{attribute 'Tc2GvlVarNames'}
VAR_GLOBAL

(*HORZ*)

	dwArm2HorzHomeStart 		: DWORD; (* %MD21900 *)
	dwArm2HorzHomeReset 		: DWORD; (* %MD21940 *)


(* xxx Horz SlantedLeft DWORD LINK with %MX21000-MX21099  xxx*)
(*======================================================*)

	dwArm2HorzStn1SlantedLeft 	: DWORD; (* %MD21004 *)
	dwArm2HorzStn2SlantedLeft 	: DWORD; (* %MD21008 *)
	dwArm2HorzStn3SlantedLeft 	: DWORD; (* %MD21012 *)
	dwArm2HorzStn4SlantedLeft 	: DWORD; (* %MD21016 *)
	dwArm2HorzStn5SlantedLeft 	: DWORD; (* %MD21020 *)
	dwArm2HorzStn6SlantedLeft 	: DWORD; (* %MD21024 *)
	dwArm2HorzStn7SlantedLeft 	: DWORD; (* %MD21028 *)
	dwArm2HorzStn8SlantedLeft 	: DWORD; (* %MD21032 *)
	dwArm2HorzStn9SlantedLeft 	: DWORD; (* %MD21036 *)
	dwArm2HorzStn10SlantedLeft 	: DWORD; (* %MD21040 *)
	dwArm2HorzStn11SlantedLeft 	: DWORD; (* %MD21044 *)
	dwArm2HorzStn12SlantedLeft 	: DWORD; (* %MD21048 *)

(* xxx Horz SlantedRight DWORD LINK with %MX21100-MX21199  xxx*)
(*======================================================*)

	dwArm2HorzStn1SlantedRight 	: DWORD; (* %MD21104 *)
	dwArm2HorzStn2SlantedRight 	: DWORD; (* %MD21108 *)
	dwArm2HorzStn3SlantedRight 	: DWORD; (* %MD21112 *)
	dwArm2HorzStn4SlantedRight 	: DWORD; (* %MD21116 *)
	dwArm2HorzStn5SlantedRight 	: DWORD; (* %MD21120 *)
	dwArm2HorzStn6SlantedRight 	: DWORD; (* %MD21124 *)
	dwArm2HorzStn7SlantedRight 	: DWORD; (* %MD21128 *)
	dwArm2HorzStn8SlantedRight 	: DWORD; (* %MD21132 *)
	dwArm2HorzStn9SlantedRight 	: DWORD; (* %MD21136 *)
	dwArm2HorzStn10SlantedRight 	: DWORD; (* %MD21140 *)
	dwArm2HorzStn11SlantedRight 	: DWORD; (* %MD21144 *)
	dwArm2HorzStn12SlantedRight 	: DWORD; (* %MD21148 *)

(* xxx Hook DWORD LINK with %MX21200-MX21299  xxx*)
(*======================================================*)

	dwArm2Ld1Hook 				: DWORD; (* %MD21252 *)
	dwArm2Uld1Hook 			: DWORD; (* %MD21256 *)
	dwArm2HorzStn1Hook 			: DWORD; (* %MD21204 *)
	dwArm2HorzStn2Hook 			: DWORD; (* %MD21208 *)
	dwArm2HorzStn3Hook 			: DWORD; (* %MD21212 *)
	dwArm2HorzStn4Hook 			: DWORD; (* %MD21216 *)
	dwArm2HorzStn5Hook 			: DWORD; (* %MD21220 *)
	dwArm2HorzStn6Hook 			: DWORD; (* %MD21224 *)
	dwArm2HorzStn7Hook 			: DWORD; (* %MD21228 *)
	dwArm2HorzStn8Hook 			: DWORD; (* %MD21232 *)
	dwArm2HorzStn9Hook 			: DWORD; (* %MD21236 *)
	dwArm2HorzStn10Hook 		: DWORD; (* %MD21240 *)
	dwArm2HorzStn11Hook 		: DWORD; (* %MD21244 *)
	dwArm2HorzStn12Hook 		: DWORD; (* %MD21248 *)

(* xxx Unhook DWORD LINK with %MX21300-MX21399  xxx*)
(*======================================================*)

	dwArm2Ld1Unhook 			: DWORD; (* %MD21352 *)
	dwArm2Uld1Unhook 			: DWORD; (* %MD21356 *)
	dwArm2HorzStn1Unhook 		: DWORD; (* %MD21304 *)
	dwArm2HorzStn2Unhook 		: DWORD; (* %MD21308 *)
	dwArm2HorzStn3Unhook 		: DWORD; (* %MD21312 *)
	dwArm2HorzStn4Unhook 		: DWORD; (* %MD21316 *)
	dwArm2HorzStn5Unhook 		: DWORD; (* %MD21320 *)
	dwArm2HorzStn6Unhook 		: DWORD; (* %MD21324 *)
	dwArm2HorzStn7Unhook 		: DWORD; (* %MD21328 *)
	dwArm2HorzStn8Unhook 		: DWORD; (* %MD21332 *)
	dwArm2HorzStn9Unhook 		: DWORD; (* %MD21336 *)
	dwArm2HorzStn10Unhook 		: DWORD; (* %MD21340 *)
	dwArm2HorzStn11Unhook 		: DWORD; (* %MD21344 *)
	dwArm2HorzStn12Unhook 		: DWORD; (* %MD21348 *)

(*VERT*)

	dwArm2VertHomeStart 			: DWORD; (* %MD26900 *)
	dwArm2VertHomeReset 		: DWORD; (* %MD26940 *)

(* xxx Up DWORD LINK with %MX26000-MX26099  xxx*)
(*======================================================*)

	dwArm2Ld1Up 				: DWORD; (* %MD26052 *)
	dwArm2Uld1Up 				: DWORD; (* %MD26056 *)
	dwArm2VertStn1Up 			: DWORD; (* %MD26004 *)
	dwArm2VertStn2Up 			: DWORD; (* %MD26008 *)
	dwArm2VertStn3Up 			: DWORD; (* %MD26012 *)
	dwArm2VertStn4Up 			: DWORD; (* %MD26016 *)
	dwArm2VertStn5Up 			: DWORD; (* %MD26020 *)
	dwArm2VertStn6Up 			: DWORD; (* %MD26024 *)
	dwArm2VertStn7Up 			: DWORD; (* %MD26028 *)
	dwArm2VertStn8Up 			: DWORD; (* %MD26032 *)
	dwArm2VertStn9Up 			: DWORD; (* %MD26036 *)
	dwArm2VertStn10Up 			: DWORD; (* %MD26040 *)
	dwArm2VertStn11Up 			: DWORD; (* %MD26044 *)
	dwArm2VertStn12Up 			: DWORD; (* %MD26048 *)

(* xxx Down SpSlanted DWORD LINK with %MX26100-MX26199  xxx*)
(*======================================================*)
(*Arm Mid Pos*)
	dwArm2VertStn1SpSlanted 		: DWORD; (* %MD26104 *)
	dwArm2VertStn2SpSlanted 		: DWORD; (* %MD26108 *)
	dwArm2VertStn3SpSlanted 		: DWORD; (* %MD26112 *)
	dwArm2VertStn4SpSlanted 		: DWORD; (* %MD26116 *)
	dwArm2VertStn5SpSlanted 		: DWORD; (* %MD26120 *)
	dwArm2VertStn6SpSlanted 		: DWORD; (* %MD26124 *)
	dwArm2VertStn7SpSlanted 		: DWORD; (* %MD26128 *)
	dwArm2VertStn8SpSlanted 		: DWORD; (* %MD26132 *)
	dwArm2VertStn9SpSlanted 		: DWORD; (* %MD26136 *)
	dwArm2VertStn10SpSlanted 	: DWORD; (* %MD26140 *)
	dwArm2VertStn11SpSlanted 	: DWORD; (* %MD26144 *)
	dwArm2VertStn12SpSlanted 	: DWORD; (* %MD26148 *)

(* xxx Down Regular DWORD LINK with %MX26200-MX26299  xxx*)
(*======================================================*)

	dwArm2VertStn1Regular 		: DWORD; (* %MD26204 *)
	dwArm2VertStn2Regular 		: DWORD; (* %MD26208 *)
	dwArm2VertStn3Regular 		: DWORD; (* %MD26212 *)
	dwArm2VertStn4Regular 		: DWORD; (* %MD26216 *)
	dwArm2VertStn5Regular 		: DWORD; (* %MD26220 *)
	dwArm2VertStn6Regular 		: DWORD; (* %MD26224 *)
	dwArm2VertStn7Regular 		: DWORD; (* %MD26228 *)
	dwArm2VertStn8Regular 		: DWORD; (* %MD26232 *)
	dwArm2VertStn9Regular 		: DWORD; (* %MD26236 *)
	dwArm2VertStn10Regular 		: DWORD; (* %MD26240 *)
	dwArm2VertStn11Regular 		: DWORD; (* %MD26244 *)
	dwArm2VertStn12Regular 		: DWORD; (* %MD26248 *)

(* xxx Up AgiUp DWORD LINK with %MX26300-MX26399  xxx*)
(*======================================================*)

	dwArm2VertStn1AglUp 			: DWORD; (* %MD26304 *)
	dwArm2VertStn2AglUp 			: DWORD; (* %MD26308 *)
	dwArm2VertStn3AglUp 			: DWORD; (* %MD26312 *)
	dwArm2VertStn4AglUp 			: DWORD; (* %MD26316 *)
	dwArm2VertStn5AglUp 			: DWORD; (* %MD26320 *)
	dwArm2VertStn6AglUp 			: DWORD; (* %MD26324 *)
	dwArm2VertStn7AglUp 			: DWORD; (* %MD26328 *)
	dwArm2VertStn8AglUp 			: DWORD; (* %MD26332 *)
	dwArm2VertStn9AglUp 			: DWORD; (* %MD26336 *)
	dwArm2VertStn10AglUp 		: DWORD; (* %MD26340 *)
	dwArm2VertStn11AglUp 		: DWORD; (* %MD26344 *)
	dwArm2VertStn12AglUp 		: DWORD; (* %MD26348 *)

(* xxx Down AgiDown DWORD LINK with %MX26400-MX26499  xxx*)
(*======================================================*)

	dwArm2VertStn1AglDown 		: DWORD; (* %MD26404 *)
	dwArm2VertStn2AglDown 		: DWORD; (* %MD26408 *)
	dwArm2VertStn3AglDown 		: DWORD; (* %MD26412 *)
	dwArm2VertStn4AglDown 		: DWORD; (* %MD26416 *)
	dwArm2VertStn5AglDown 		: DWORD; (* %MD26420 *)
	dwArm2VertStn6AglDown 		: DWORD; (* %MD26424 *)
	dwArm2VertStn7AglDown 		: DWORD; (* %MD26428 *)
	dwArm2VertStn8AglDown 		: DWORD; (* %MD26432 *)
	dwArm2VertStn9AglDown 		: DWORD; (* %MD26436 *)
	dwArm2VertStn10AglDown 		: DWORD; (* %MD26440 *)
	dwArm2VertStn11AglDown 		: DWORD; (* %MD26444 *)
	dwArm2VertStn12AglDown 		: DWORD; (* %MD26448 *)

(* xxx Down DWORD LINK with %MX26500-MX26599  xxx*)
(*======================================================*)

	dwArm2Ld1Down 				: DWORD; (* %MD26552 *)
	dwArm2Uld1Down 			: DWORD; (* %MD26556 *)
	dwArm2VertStn1Down 			: DWORD; (* %MD26504 *)
	dwArm2VertStn2Down 			: DWORD; (* %MD26508 *)
	dwArm2VertStn3Down 			: DWORD; (* %MD26512 *)
	dwArm2VertStn4Down 			: DWORD; (* %MD26516 *)
	dwArm2VertStn5Down 			: DWORD; (* %MD26520 *)
	dwArm2VertStn6Down 			: DWORD; (* %MD26524 *)
	dwArm2VertStn7Down 			: DWORD; (* %MD26528 *)
	dwArm2VertStn8Down 			: DWORD; (* %MD26532 *)
	dwArm2VertStn9Down 			: DWORD; (* %MD26536 *)
	dwArm2VertStn10Down 		: DWORD; (* %MD26540 *)
	dwArm2VertStn11Down 		: DWORD; (* %MD26544 *)
	dwArm2VertStn12Down 		: DWORD; (* %MD26548 *)

(*LIFTER*)

	dwSlowPull2LifterHomeStart 	: DWORD; (* %MD31900 *)
	dwSlowPull2LifterHomeReset 	: DWORD; (* %MD31940 *)

(* xxx Up/Down LifterUp DWORD LINK with %MX31000-   xxx*)
(*======================================================*)

	dwSlowPull2LifterStn1Up 		: DWORD; (* %MD31004 *)
	dwSlowPull2LifterStn2Up 		: DWORD; (* %MD31008 *)
	dwSlowPull2LifterStn3Up 		: DWORD; (* %MD31012 *)
	dwSlowPull2LifterStn4Up 		: DWORD; (* %MD31016 *)
	dwSlowPull2LifterStn5Up 		: DWORD; (* %MD31020 *)
	dwSlowPull2LifterStn6Up 		: DWORD; (* %MD31024 *)
	dwSlowPull2LifterStn7Up 		: DWORD; (* %MD31028 *)
	dwSlowPull2LifterStn8Up 		: DWORD; (* %MD31032 *)
	dwSlowPull2LifterStn9Up 		: DWORD; (* %MD31036 *)
	dwSlowPull2LifterStn10Up 		: DWORD; (* %MD31040 *)
	dwSlowPull2LifterStn11Up 		: DWORD; (* %MD31044 *)
	dwSlowPull2LifterStn12Up 		: DWORD; (* %MD31048 *)

(* xxx Up/Down LifterDown DWORD LINK with %MX31000-   xxx*)
(*======================================================*)

	dwSlowPull2LifterStn1Down 		: DWORD; (* %MD31304 *)
	dwSlowPull2LifterStn2Down 		: DWORD; (* %MD31308 *)
	dwSlowPull2LifterStn3Down 		: DWORD; (* %MD31312 *)
	dwSlowPull2LifterStn4Down 		: DWORD; (* %MD31316 *)
	dwSlowPull2LifterStn5Down 		: DWORD; (* %MD31320 *)
	dwSlowPull2LifterStn6Down 		: DWORD; (* %MD31324 *)
	dwSlowPull2LifterStn7Down 		: DWORD; (* %MD31328 *)
	dwSlowPull2LifterStn8Down 		: DWORD; (* %MD31332 *)
	dwSlowPull2LifterStn9Down 		: DWORD; (* %MD31336 *)
	dwSlowPull2LifterStn10Down 	: DWORD; (* %MD31340 *)
	dwSlowPull2LifterStn11Down 	: DWORD; (* %MD31344 *)
	dwSlowPull2LifterStn12Down 	: DWORD; (* %MD31348 *)

(* xxx Up/Down LifterAgiUp DWORD LINK with %MX31000-   xxx*)
(*======================================================*)

	dwSlowPull2LifterStn1AgiUp 	: DWORD; (* %MD31104 *)
	dwSlowPull2LifterStn2AgiUp 	: DWORD; (* %MD31108 *)
	dwSlowPull2LifterStn3AgiUp 	: DWORD; (* %MD31112 *)
	dwSlowPull2LifterStn4AgiUp 	: DWORD; (* %MD31116 *)
	dwSlowPull2LifterStn5AgiUp 	: DWORD; (* %MD31120 *)
	dwSlowPull2LifterStn6AgiUp 	: DWORD; (* %MD31124 *)
	dwSlowPull2LifterStn7AgiUp 	: DWORD; (* %MD31128 *)
	dwSlowPull2LifterStn8AgiUp 	: DWORD; (* %MD31132 *)
	dwSlowPull2LifterStn9AgiUp 	: DWORD; (* %MD31136 *)
	dwSlowPull2LifterStn10AgiUp 	: DWORD; (* %MD31140 *)
	dwSlowPull2LifterStn11AgiUp 	: DWORD; (* %MD31144 *)
	dwSlowPull2LifterStn12AgiUp 	: DWORD; (* %MD31148 *)

(* xxx Up/Down LifterAgiDown DWORD LINK with %MX31000-   xxx*)
(*======================================================*)

	dwSlowPull2LifterStn1AgiDown 	: DWORD; (* %MD31204 *)
	dwSlowPull2LifterStn2AgiDown 	: DWORD; (* %MD31208 *)
	dwSlowPull2LifterStn3AgiDown 	: DWORD; (* %MD31212 *)
	dwSlowPull2LifterStn4AgiDown 	: DWORD; (* %MD31216 *)
	dwSlowPull2LifterStn5AgiDown 	: DWORD; (* %MD31220 *)
	dwSlowPull2LifterStn6AgiDown 	: DWORD; (* %MD31224 *)
	dwSlowPull2LifterStn7AgiDown 	: DWORD; (* %MD31228 *)
	dwSlowPull2LifterStn8AgiDown 	: DWORD; (* %MD31232 *)
	dwSlowPull2LifterStn9AgiDown 	: DWORD; (* %MD31236 *)
	dwSlowPull2LifterStn10AgiDown 	: DWORD; (* %MD31240 *)
	dwSlowPull2LifterStn11AgiDown 	: DWORD; (* %MD31244 *)
	dwSlowPull2LifterStn12AgiDown 	: DWORD; (* %MD31248 *)

(* xxxxxxxxxxxxxxxxxxxxxxxxxxxxxxxxxxxxxxx Home xxxxxxxxxxxxxxxxxxxxxxxxxxxxxxxxxxxxxxx*)
(*====================== Vert Home BOOL LINK with %MX26900 ======================*)

	bArm2VertHomeStart_00 AT %MX26900.0 : BOOL;
	bArm2VertHomeStart_01 AT %MX26900.1 : BOOL;
	bArm2VertHomeStart_02 AT %MX26900.2 : BOOL;
	bArm2VertHomeStart_03 AT %MX26900.3 : BOOL;
	bArm2VertHomeStart_04 AT %MX26900.4 : BOOL;
	bArm2VertHomeStart_05 AT %MX26900.5 : BOOL;
	bArm2VertHomeStart_06 AT %MX26900.6 : BOOL;
	bArm2VertHomeStart_07 AT %MX26900.7 : BOOL;
	bArm2VertHomeStart_08 AT %MX26900.8 : BOOL;
	bArm2VertHomeStart_09 AT %MX26900.9 : BOOL;
	bArm2VertHomeStart_10 AT %MX26900.10 : BOOL;
	bArm2VertHomeStart_11 AT %MX26900.11 : BOOL;
	bArm2VertHomeStart_12 AT %MX26900.12 : BOOL;
	bArm2VertHomeStart_13 AT %MX26900.13 : BOOL;
	bArm2VertHomeStart_14 AT %MX26900.14 : BOOL;
	bArm2VertHomeStart_15 AT %MX26900.15 : BOOL;
	bArm2VertHomeStart_16 AT %MX26900.16 : BOOL;
	bArm2VertHomeStart_17 AT %MX26900.17 : BOOL;
	bArm2VertHomeStart_18 AT %MX26900.18 : BOOL;
	bArm2VertHomeStart_19 AT %MX26900.19 : BOOL;
	bArm2VertHomeStart_20 AT %MX26900.20 : BOOL;
	bArm2VertHomeStart_21 AT %MX26900.21 : BOOL;
	bArm2VertHomeStart_22 AT %MX26900.22 : BOOL;
	bArm2VertHomeStart_23 AT %MX26900.23 : BOOL;
	bArm2VertHomeStart_24 AT %MX26900.24 : BOOL;
	bArm2VertHomeStart_25 AT %MX26900.25 : BOOL;
	bArm2VertHomeStart_26 AT %MX26900.26 : BOOL;
	bArm2VertHomeStart_27 AT %MX26900.27 : BOOL;
	bArm2VertHomeStart_28 AT %MX26900.28 : BOOL;
	bArm2VertHomeStart_29 AT %MX26900.29 : BOOL;
	bArm2VertHomeStart_30 AT %MX26900.30 : BOOL;
	bArm2VertHomeStart_31 AT %MX26900.31 : BOOL;

	bArm2HorzHomeStart_00 AT %MX21900.0 : BOOL;
	bArm2HorzHomeStart_01 AT %MX21900.1 : BOOL;
	bArm2HorzHomeStart_02 AT %MX21900.2 : BOOL;
	bArm2HorzHomeStart_03 AT %MX21900.3 : BOOL;
	bArm2HorzHomeStart_04 AT %MX21900.4 : BOOL;
	bArm2HorzHomeStart_05 AT %MX21900.5 : BOOL;
	bArm2HorzHomeStart_06 AT %MX21900.6 : BOOL;
	bArm2HorzHomeStart_07 AT %MX21900.7 : BOOL;
	bArm2HorzHomeStart_08 AT %MX21900.8 : BOOL;
	bArm2HorzHomeStart_09 AT %MX21900.9 : BOOL;
	bArm2HorzHomeStart_10 AT %MX21900.10 : BOOL;
	bArm2HorzHomeStart_11 AT %MX21900.11 : BOOL;
	bArm2HorzHomeStart_12 AT %MX21900.12 : BOOL;
	bArm2HorzHomeStart_13 AT %MX21900.13 : BOOL;
	bArm2HorzHomeStart_14 AT %MX21900.14 : BOOL;
	bArm2HorzHomeStart_15 AT %MX21900.15 : BOOL;
	bArm2HorzHomeStart_16 AT %MX21900.16 : BOOL;
	bArm2HorzHomeStart_17 AT %MX21900.17 : BOOL;
	bArm2HorzHomeStart_18 AT %MX21900.18 : BOOL;
	bArm2HorzHomeStart_19 AT %MX21900.19 : BOOL;
	bArm2HorzHomeStart_20 AT %MX21900.20 : BOOL;
	bArm2HorzHomeStart_21 AT %MX21900.21 : BOOL;
	bArm2HorzHomeStart_22 AT %MX21900.22 : BOOL;
	bArm2HorzHomeStart_23 AT %MX21900.23 : BOOL;
	bArm2HorzHomeStart_24 AT %MX21900.24 : BOOL;
	bArm2HorzHomeStart_25 AT %MX21900.25 : BOOL;
	bArm2HorzHomeStart_26 AT %MX21900.26 : BOOL;
	bArm2HorzHomeStart_27 AT %MX21900.27 : BOOL;
	bArm2HorzHomeStart_28 AT %MX21900.28 : BOOL;
	bArm2HorzHomeStart_29 AT %MX21900.29 : BOOL;
	bArm2HorzHomeStart_30 AT %MX21900.30 : BOOL;
	bArm2HorzHomeStart_31 AT %MX21900.31 : BOOL;

	bSlowPull2LifterHomeStart_00 AT %MX31900.0 : BOOL;
	bSlowPull2LifterHomeStart_01 AT %MX31900.1 : BOOL;
	bSlowPull2LifterHomeStart_02 AT %MX31900.2 : BOOL;
	bSlowPull2LifterHomeStart_03 AT %MX31900.3 : BOOL;
	bSlowPull2LifterHomeStart_04 AT %MX31900.4 : BOOL;
	bSlowPull2LifterHomeStart_05 AT %MX31900.5 : BOOL;
	bSlowPull2LifterHomeStart_06 AT %MX31900.6 : BOOL;
	bSlowPull2LifterHomeStart_07 AT %MX31900.7 : BOOL;
	bSlowPull2LifterHomeStart_08 AT %MX31900.8 : BOOL;
	bSlowPull2LifterHomeStart_09 AT %MX31900.9 : BOOL;
	bSlowPull2LifterHomeStart_10 AT %MX31900.10 : BOOL;
	bSlowPull2LifterHomeStart_11 AT %MX31900.11 : BOOL;
	bSlowPull2LifterHomeStart_12 AT %MX31900.12 : BOOL;
	bSlowPull2LifterHomeStart_13 AT %MX31900.13 : BOOL;
	bSlowPull2LifterHomeStart_14 AT %MX31900.14 : BOOL;
	bSlowPull2LifterHomeStart_15 AT %MX31900.15 : BOOL;
	bSlowPull2LifterHomeStart_16 AT %MX31900.16 : BOOL;
	bSlowPull2LifterHomeStart_17 AT %MX31900.17 : BOOL;
	bSlowPull2LifterHomeStart_18 AT %MX31900.18 : BOOL;
	bSlowPull2LifterHomeStart_19 AT %MX31900.19 : BOOL;
	bSlowPull2LifterHomeStart_20 AT %MX31900.20 : BOOL;
	bSlowPull2LifterHomeStart_21 AT %MX31900.21 : BOOL;
	bSlowPull2LifterHomeStart_22 AT %MX31900.22 : BOOL;
	bSlowPull2LifterHomeStart_23 AT %MX31900.23 : BOOL;
	bSlowPull2LifterHomeStart_24 AT %MX31900.24 : BOOL;
	bSlowPull2LifterHomeStart_25 AT %MX31900.25 : BOOL;
	bSlowPull2LifterHomeStart_26 AT %MX31900.26 : BOOL;
	bSlowPull2LifterHomeStart_27 AT %MX31900.27 : BOOL;
	bSlowPull2LifterHomeStart_28 AT %MX31900.28 : BOOL;
	bSlowPull2LifterHomeStart_29 AT %MX31900.29 : BOOL;
	bSlowPull2LifterHomeStart_30 AT %MX31900.30 : BOOL;
	bSlowPull2LifterHomeStart_31 AT %MX31900.31 : BOOL;

(*=============================== SlantedLeft word ===============================*)
(*====================== SlantedLeft BOOL LINK with %MX21000-MX21099 ======================*)

	bArm2HorzStn1SlantedLeft_00 AT %MX21004.0 : BOOL;
	bArm2HorzStn1SlantedLeft_01 AT %MX21004.1 : BOOL;
	bArm2HorzStn1SlantedLeft_02 AT %MX21004.2 : BOOL;
	bArm2HorzStn1SlantedLeft_03 AT %MX21004.3 : BOOL;
	bArm2HorzStn1SlantedLeft_04 AT %MX21004.4 : BOOL;
	bArm2HorzStn1SlantedLeft_05 AT %MX21004.5 : BOOL;
	bArm2HorzStn1SlantedLeft_06 AT %MX21004.6 : BOOL;
	bArm2HorzStn1SlantedLeft_07 AT %MX21004.7 : BOOL;
	bArm2HorzStn1SlantedLeft_08 AT %MX21004.8 : BOOL;
	bArm2HorzStn1SlantedLeft_09 AT %MX21004.9 : BOOL;
	bArm2HorzStn1SlantedLeft_10 AT %MX21004.10 : BOOL;
	bArm2HorzStn1SlantedLeft_11 AT %MX21004.11 : BOOL;
	bArm2HorzStn1SlantedLeft_12 AT %MX21004.12 : BOOL;
	bArm2HorzStn1SlantedLeft_13 AT %MX21004.13 : BOOL;
	bArm2HorzStn1SlantedLeft_14 AT %MX21004.14 : BOOL;
	bArm2HorzStn1SlantedLeft_15 AT %MX21004.15 : BOOL;
	bArm2HorzStn1SlantedLeft_16 AT %MX21004.16 : BOOL;
	bArm2HorzStn1SlantedLeft_17 AT %MX21004.17 : BOOL;
	bArm2HorzStn1SlantedLeft_18 AT %MX21004.18 : BOOL;
	bArm2HorzStn1SlantedLeft_19 AT %MX21004.19 : BOOL;
	bArm2HorzStn1SlantedLeft_20 AT %MX21004.20 : BOOL;
	bArm2HorzStn1SlantedLeft_21 AT %MX21004.21 : BOOL;
	bArm2HorzStn1SlantedLeft_22 AT %MX21004.22 : BOOL;
	bArm2HorzStn1SlantedLeft_23 AT %MX21004.23 : BOOL;
	bArm2HorzStn1SlantedLeft_24 AT %MX21004.24 : BOOL;
	bArm2HorzStn1SlantedLeft_25 AT %MX21004.25 : BOOL;
	bArm2HorzStn1SlantedLeft_26 AT %MX21004.26 : BOOL;
	bArm2HorzStn1SlantedLeft_27 AT %MX21004.27 : BOOL;
	bArm2HorzStn1SlantedLeft_28 AT %MX21004.28 : BOOL;
	bArm2HorzStn1SlantedLeft_29 AT %MX21004.29 : BOOL;
	bArm2HorzStn1SlantedLeft_30 AT %MX21004.30 : BOOL;
	bArm2HorzStn1SlantedLeft_31 AT %MX21004.31 : BOOL;

	bArm2HorzStn2SlantedLeft_00 AT %MX21008.0 : BOOL;
	bArm2HorzStn2SlantedLeft_01 AT %MX21008.1 : BOOL;
	bArm2HorzStn2SlantedLeft_02 AT %MX21008.2 : BOOL;
	bArm2HorzStn2SlantedLeft_03 AT %MX21008.3 : BOOL;
	bArm2HorzStn2SlantedLeft_04 AT %MX21008.4 : BOOL;
	bArm2HorzStn2SlantedLeft_05 AT %MX21008.5 : BOOL;
	bArm2HorzStn2SlantedLeft_06 AT %MX21008.6 : BOOL;
	bArm2HorzStn2SlantedLeft_07 AT %MX21008.7 : BOOL;
	bArm2HorzStn2SlantedLeft_08 AT %MX21008.8 : BOOL;
	bArm2HorzStn2SlantedLeft_09 AT %MX21008.9 : BOOL;
	bArm2HorzStn2SlantedLeft_10 AT %MX21008.10 : BOOL;
	bArm2HorzStn2SlantedLeft_11 AT %MX21008.11 : BOOL;
	bArm2HorzStn2SlantedLeft_12 AT %MX21008.12 : BOOL;
	bArm2HorzStn2SlantedLeft_13 AT %MX21008.13 : BOOL;
	bArm2HorzStn2SlantedLeft_14 AT %MX21008.14 : BOOL;
	bArm2HorzStn2SlantedLeft_15 AT %MX21008.15 : BOOL;
	bArm2HorzStn2SlantedLeft_16 AT %MX21008.16 : BOOL;
	bArm2HorzStn2SlantedLeft_17 AT %MX21008.17 : BOOL;
	bArm2HorzStn2SlantedLeft_18 AT %MX21008.18 : BOOL;
	bArm2HorzStn2SlantedLeft_19 AT %MX21008.19 : BOOL;
	bArm2HorzStn2SlantedLeft_20 AT %MX21008.20 : BOOL;
	bArm2HorzStn2SlantedLeft_21 AT %MX21008.21 : BOOL;
	bArm2HorzStn2SlantedLeft_22 AT %MX21008.22 : BOOL;
	bArm2HorzStn2SlantedLeft_23 AT %MX21008.23 : BOOL;
	bArm2HorzStn2SlantedLeft_24 AT %MX21008.24 : BOOL;
	bArm2HorzStn2SlantedLeft_25 AT %MX21008.25 : BOOL;
	bArm2HorzStn2SlantedLeft_26 AT %MX21008.26 : BOOL;
	bArm2HorzStn2SlantedLeft_27 AT %MX21008.27 : BOOL;
	bArm2HorzStn2SlantedLeft_28 AT %MX21008.28 : BOOL;
	bArm2HorzStn2SlantedLeft_29 AT %MX21008.29 : BOOL;
	bArm2HorzStn2SlantedLeft_30 AT %MX21008.30 : BOOL;
	bArm2HorzStn2SlantedLeft_31 AT %MX21008.31 : BOOL;

	bArm2HorzStn3SlantedLeft_00 AT %MX21012.0 : BOOL;
	bArm2HorzStn3SlantedLeft_01 AT %MX21012.1 : BOOL;
	bArm2HorzStn3SlantedLeft_02 AT %MX21012.2 : BOOL;
	bArm2HorzStn3SlantedLeft_03 AT %MX21012.3 : BOOL;
	bArm2HorzStn3SlantedLeft_04 AT %MX21012.4 : BOOL;
	bArm2HorzStn3SlantedLeft_05 AT %MX21012.5 : BOOL;
	bArm2HorzStn3SlantedLeft_06 AT %MX21012.6 : BOOL;
	bArm2HorzStn3SlantedLeft_07 AT %MX21012.7 : BOOL;
	bArm2HorzStn3SlantedLeft_08 AT %MX21012.8 : BOOL;
	bArm2HorzStn3SlantedLeft_09 AT %MX21012.9 : BOOL;
	bArm2HorzStn3SlantedLeft_10 AT %MX21012.10 : BOOL;
	bArm2HorzStn3SlantedLeft_11 AT %MX21012.11 : BOOL;
	bArm2HorzStn3SlantedLeft_12 AT %MX21012.12 : BOOL;
	bArm2HorzStn3SlantedLeft_13 AT %MX21012.13 : BOOL;
	bArm2HorzStn3SlantedLeft_14 AT %MX21012.14 : BOOL;
	bArm2HorzStn3SlantedLeft_15 AT %MX21012.15 : BOOL;
	bArm2HorzStn3SlantedLeft_16 AT %MX21012.16 : BOOL;
	bArm2HorzStn3SlantedLeft_17 AT %MX21012.17 : BOOL;
	bArm2HorzStn3SlantedLeft_18 AT %MX21012.18 : BOOL;
	bArm2HorzStn3SlantedLeft_19 AT %MX21012.19 : BOOL;
	bArm2HorzStn3SlantedLeft_20 AT %MX21012.20 : BOOL;
	bArm2HorzStn3SlantedLeft_21 AT %MX21012.21 : BOOL;
	bArm2HorzStn3SlantedLeft_22 AT %MX21012.22 : BOOL;
	bArm2HorzStn3SlantedLeft_23 AT %MX21012.23 : BOOL;
	bArm2HorzStn3SlantedLeft_24 AT %MX21012.24 : BOOL;
	bArm2HorzStn3SlantedLeft_25 AT %MX21012.25 : BOOL;
	bArm2HorzStn3SlantedLeft_26 AT %MX21012.26 : BOOL;
	bArm2HorzStn3SlantedLeft_27 AT %MX21012.27 : BOOL;
	bArm2HorzStn3SlantedLeft_28 AT %MX21012.28 : BOOL;
	bArm2HorzStn3SlantedLeft_29 AT %MX21012.29 : BOOL;
	bArm2HorzStn3SlantedLeft_30 AT %MX21012.30 : BOOL;
	bArm2HorzStn3SlantedLeft_31 AT %MX21012.31 : BOOL;

	bArm2HorzStn4SlantedLeft_00 AT %MX21016.0 : BOOL;
	bArm2HorzStn4SlantedLeft_01 AT %MX21016.1 : BOOL;
	bArm2HorzStn4SlantedLeft_02 AT %MX21016.2 : BOOL;
	bArm2HorzStn4SlantedLeft_03 AT %MX21016.3 : BOOL;
	bArm2HorzStn4SlantedLeft_04 AT %MX21016.4 : BOOL;
	bArm2HorzStn4SlantedLeft_05 AT %MX21016.5 : BOOL;
	bArm2HorzStn4SlantedLeft_06 AT %MX21016.6 : BOOL;
	bArm2HorzStn4SlantedLeft_07 AT %MX21016.7 : BOOL;
	bArm2HorzStn4SlantedLeft_08 AT %MX21016.8 : BOOL;
	bArm2HorzStn4SlantedLeft_09 AT %MX21016.9 : BOOL;
	bArm2HorzStn4SlantedLeft_10 AT %MX21016.10 : BOOL;
	bArm2HorzStn4SlantedLeft_11 AT %MX21016.11 : BOOL;
	bArm2HorzStn4SlantedLeft_12 AT %MX21016.12 : BOOL;
	bArm2HorzStn4SlantedLeft_13 AT %MX21016.13 : BOOL;
	bArm2HorzStn4SlantedLeft_14 AT %MX21016.14 : BOOL;
	bArm2HorzStn4SlantedLeft_15 AT %MX21016.15 : BOOL;
	bArm2HorzStn4SlantedLeft_16 AT %MX21016.16 : BOOL;
	bArm2HorzStn4SlantedLeft_17 AT %MX21016.17 : BOOL;
	bArm2HorzStn4SlantedLeft_18 AT %MX21016.18 : BOOL;
	bArm2HorzStn4SlantedLeft_19 AT %MX21016.19 : BOOL;
	bArm2HorzStn4SlantedLeft_20 AT %MX21016.20 : BOOL;
	bArm2HorzStn4SlantedLeft_21 AT %MX21016.21 : BOOL;
	bArm2HorzStn4SlantedLeft_22 AT %MX21016.22 : BOOL;
	bArm2HorzStn4SlantedLeft_23 AT %MX21016.23 : BOOL;
	bArm2HorzStn4SlantedLeft_24 AT %MX21016.24 : BOOL;
	bArm2HorzStn4SlantedLeft_25 AT %MX21016.25 : BOOL;
	bArm2HorzStn4SlantedLeft_26 AT %MX21016.26 : BOOL;
	bArm2HorzStn4SlantedLeft_27 AT %MX21016.27 : BOOL;
	bArm2HorzStn4SlantedLeft_28 AT %MX21016.28 : BOOL;
	bArm2HorzStn4SlantedLeft_29 AT %MX21016.29 : BOOL;
	bArm2HorzStn4SlantedLeft_30 AT %MX21016.30 : BOOL;
	bArm2HorzStn4SlantedLeft_31 AT %MX21016.31 : BOOL;

	bArm2HorzStn5SlantedLeft_00 AT %MX21020.0 : BOOL;
	bArm2HorzStn5SlantedLeft_01 AT %MX21020.1 : BOOL;
	bArm2HorzStn5SlantedLeft_02 AT %MX21020.2 : BOOL;
	bArm2HorzStn5SlantedLeft_03 AT %MX21020.3 : BOOL;
	bArm2HorzStn5SlantedLeft_04 AT %MX21020.4 : BOOL;
	bArm2HorzStn5SlantedLeft_05 AT %MX21020.5 : BOOL;
	bArm2HorzStn5SlantedLeft_06 AT %MX21020.6 : BOOL;
	bArm2HorzStn5SlantedLeft_07 AT %MX21020.7 : BOOL;
	bArm2HorzStn5SlantedLeft_08 AT %MX21020.8 : BOOL;
	bArm2HorzStn5SlantedLeft_09 AT %MX21020.9 : BOOL;
	bArm2HorzStn5SlantedLeft_10 AT %MX21020.10 : BOOL;
	bArm2HorzStn5SlantedLeft_11 AT %MX21020.11 : BOOL;
	bArm2HorzStn5SlantedLeft_12 AT %MX21020.12 : BOOL;
	bArm2HorzStn5SlantedLeft_13 AT %MX21020.13 : BOOL;
	bArm2HorzStn5SlantedLeft_14 AT %MX21020.14 : BOOL;
	bArm2HorzStn5SlantedLeft_15 AT %MX21020.15 : BOOL;
	bArm2HorzStn5SlantedLeft_16 AT %MX21020.16 : BOOL;
	bArm2HorzStn5SlantedLeft_17 AT %MX21020.17 : BOOL;
	bArm2HorzStn5SlantedLeft_18 AT %MX21020.18 : BOOL;
	bArm2HorzStn5SlantedLeft_19 AT %MX21020.19 : BOOL;
	bArm2HorzStn5SlantedLeft_20 AT %MX21020.20 : BOOL;
	bArm2HorzStn5SlantedLeft_21 AT %MX21020.21 : BOOL;
	bArm2HorzStn5SlantedLeft_22 AT %MX21020.22 : BOOL;
	bArm2HorzStn5SlantedLeft_23 AT %MX21020.23 : BOOL;
	bArm2HorzStn5SlantedLeft_24 AT %MX21020.24 : BOOL;
	bArm2HorzStn5SlantedLeft_25 AT %MX21020.25 : BOOL;
	bArm2HorzStn5SlantedLeft_26 AT %MX21020.26 : BOOL;
	bArm2HorzStn5SlantedLeft_27 AT %MX21020.27 : BOOL;
	bArm2HorzStn5SlantedLeft_28 AT %MX21020.28 : BOOL;
	bArm2HorzStn5SlantedLeft_29 AT %MX21020.29 : BOOL;
	bArm2HorzStn5SlantedLeft_30 AT %MX21020.30 : BOOL;
	bArm2HorzStn5SlantedLeft_31 AT %MX21020.31 : BOOL;

	bArm2HorzStn6SlantedLeft_00 AT %MX21024.0 : BOOL;
	bArm2HorzStn6SlantedLeft_01 AT %MX21024.1 : BOOL;
	bArm2HorzStn6SlantedLeft_02 AT %MX21024.2 : BOOL;
	bArm2HorzStn6SlantedLeft_03 AT %MX21024.3 : BOOL;
	bArm2HorzStn6SlantedLeft_04 AT %MX21024.4 : BOOL;
	bArm2HorzStn6SlantedLeft_05 AT %MX21024.5 : BOOL;
	bArm2HorzStn6SlantedLeft_06 AT %MX21024.6 : BOOL;
	bArm2HorzStn6SlantedLeft_07 AT %MX21024.7 : BOOL;
	bArm2HorzStn6SlantedLeft_08 AT %MX21024.8 : BOOL;
	bArm2HorzStn6SlantedLeft_09 AT %MX21024.9 : BOOL;
	bArm2HorzStn6SlantedLeft_10 AT %MX21024.10 : BOOL;
	bArm2HorzStn6SlantedLeft_11 AT %MX21024.11 : BOOL;
	bArm2HorzStn6SlantedLeft_12 AT %MX21024.12 : BOOL;
	bArm2HorzStn6SlantedLeft_13 AT %MX21024.13 : BOOL;
	bArm2HorzStn6SlantedLeft_14 AT %MX21024.14 : BOOL;
	bArm2HorzStn6SlantedLeft_15 AT %MX21024.15 : BOOL;
	bArm2HorzStn6SlantedLeft_16 AT %MX21024.16 : BOOL;
	bArm2HorzStn6SlantedLeft_17 AT %MX21024.17 : BOOL;
	bArm2HorzStn6SlantedLeft_18 AT %MX21024.18 : BOOL;
	bArm2HorzStn6SlantedLeft_19 AT %MX21024.19 : BOOL;
	bArm2HorzStn6SlantedLeft_20 AT %MX21024.20 : BOOL;
	bArm2HorzStn6SlantedLeft_21 AT %MX21024.21 : BOOL;
	bArm2HorzStn6SlantedLeft_22 AT %MX21024.22 : BOOL;
	bArm2HorzStn6SlantedLeft_23 AT %MX21024.23 : BOOL;
	bArm2HorzStn6SlantedLeft_24 AT %MX21024.24 : BOOL;
	bArm2HorzStn6SlantedLeft_25 AT %MX21024.25 : BOOL;
	bArm2HorzStn6SlantedLeft_26 AT %MX21024.26 : BOOL;
	bArm2HorzStn6SlantedLeft_27 AT %MX21024.27 : BOOL;
	bArm2HorzStn6SlantedLeft_28 AT %MX21024.28 : BOOL;
	bArm2HorzStn6SlantedLeft_29 AT %MX21024.29 : BOOL;
	bArm2HorzStn6SlantedLeft_30 AT %MX21024.30 : BOOL;
	bArm2HorzStn6SlantedLeft_31 AT %MX21024.31 : BOOL;

	bArm2HorzStn7SlantedLeft_00 AT %MX21028.0 : BOOL;
	bArm2HorzStn7SlantedLeft_01 AT %MX21028.1 : BOOL;
	bArm2HorzStn7SlantedLeft_02 AT %MX21028.2 : BOOL;
	bArm2HorzStn7SlantedLeft_03 AT %MX21028.3 : BOOL;
	bArm2HorzStn7SlantedLeft_04 AT %MX21028.4 : BOOL;
	bArm2HorzStn7SlantedLeft_05 AT %MX21028.5 : BOOL;
	bArm2HorzStn7SlantedLeft_06 AT %MX21028.6 : BOOL;
	bArm2HorzStn7SlantedLeft_07 AT %MX21028.7 : BOOL;
	bArm2HorzStn7SlantedLeft_08 AT %MX21028.8 : BOOL;
	bArm2HorzStn7SlantedLeft_09 AT %MX21028.9 : BOOL;
	bArm2HorzStn7SlantedLeft_10 AT %MX21028.10 : BOOL;
	bArm2HorzStn7SlantedLeft_11 AT %MX21028.11 : BOOL;
	bArm2HorzStn7SlantedLeft_12 AT %MX21028.12 : BOOL;
	bArm2HorzStn7SlantedLeft_13 AT %MX21028.13 : BOOL;
	bArm2HorzStn7SlantedLeft_14 AT %MX21028.14 : BOOL;
	bArm2HorzStn7SlantedLeft_15 AT %MX21028.15 : BOOL;
	bArm2HorzStn7SlantedLeft_16 AT %MX21028.16 : BOOL;
	bArm2HorzStn7SlantedLeft_17 AT %MX21028.17 : BOOL;
	bArm2HorzStn7SlantedLeft_18 AT %MX21028.18 : BOOL;
	bArm2HorzStn7SlantedLeft_19 AT %MX21028.19 : BOOL;
	bArm2HorzStn7SlantedLeft_20 AT %MX21028.20 : BOOL;
	bArm2HorzStn7SlantedLeft_21 AT %MX21028.21 : BOOL;
	bArm2HorzStn7SlantedLeft_22 AT %MX21028.22 : BOOL;
	bArm2HorzStn7SlantedLeft_23 AT %MX21028.23 : BOOL;
	bArm2HorzStn7SlantedLeft_24 AT %MX21028.24 : BOOL;
	bArm2HorzStn7SlantedLeft_25 AT %MX21028.25 : BOOL;
	bArm2HorzStn7SlantedLeft_26 AT %MX21028.26 : BOOL;
	bArm2HorzStn7SlantedLeft_27 AT %MX21028.27 : BOOL;
	bArm2HorzStn7SlantedLeft_28 AT %MX21028.28 : BOOL;
	bArm2HorzStn7SlantedLeft_29 AT %MX21028.29 : BOOL;
	bArm2HorzStn7SlantedLeft_30 AT %MX21028.30 : BOOL;
	bArm2HorzStn7SlantedLeft_31 AT %MX21028.31 : BOOL;

	bArm2HorzStn8SlantedLeft_00 AT %MX21032.0 : BOOL;
	bArm2HorzStn8SlantedLeft_01 AT %MX21032.1 : BOOL;
	bArm2HorzStn8SlantedLeft_02 AT %MX21032.2 : BOOL;
	bArm2HorzStn8SlantedLeft_03 AT %MX21032.3 : BOOL;
	bArm2HorzStn8SlantedLeft_04 AT %MX21032.4 : BOOL;
	bArm2HorzStn8SlantedLeft_05 AT %MX21032.5 : BOOL;
	bArm2HorzStn8SlantedLeft_06 AT %MX21032.6 : BOOL;
	bArm2HorzStn8SlantedLeft_07 AT %MX21032.7 : BOOL;
	bArm2HorzStn8SlantedLeft_08 AT %MX21032.8 : BOOL;
	bArm2HorzStn8SlantedLeft_09 AT %MX21032.9 : BOOL;
	bArm2HorzStn8SlantedLeft_10 AT %MX21032.10 : BOOL;
	bArm2HorzStn8SlantedLeft_11 AT %MX21032.11 : BOOL;
	bArm2HorzStn8SlantedLeft_12 AT %MX21032.12 : BOOL;
	bArm2HorzStn8SlantedLeft_13 AT %MX21032.13 : BOOL;
	bArm2HorzStn8SlantedLeft_14 AT %MX21032.14 : BOOL;
	bArm2HorzStn8SlantedLeft_15 AT %MX21032.15 : BOOL;
	bArm2HorzStn8SlantedLeft_16 AT %MX21032.16 : BOOL;
	bArm2HorzStn8SlantedLeft_17 AT %MX21032.17 : BOOL;
	bArm2HorzStn8SlantedLeft_18 AT %MX21032.18 : BOOL;
	bArm2HorzStn8SlantedLeft_19 AT %MX21032.19 : BOOL;
	bArm2HorzStn8SlantedLeft_20 AT %MX21032.20 : BOOL;
	bArm2HorzStn8SlantedLeft_21 AT %MX21032.21 : BOOL;
	bArm2HorzStn8SlantedLeft_22 AT %MX21032.22 : BOOL;
	bArm2HorzStn8SlantedLeft_23 AT %MX21032.23 : BOOL;
	bArm2HorzStn8SlantedLeft_24 AT %MX21032.24 : BOOL;
	bArm2HorzStn8SlantedLeft_25 AT %MX21032.25 : BOOL;
	bArm2HorzStn8SlantedLeft_26 AT %MX21032.26 : BOOL;
	bArm2HorzStn8SlantedLeft_27 AT %MX21032.27 : BOOL;
	bArm2HorzStn8SlantedLeft_28 AT %MX21032.28 : BOOL;
	bArm2HorzStn8SlantedLeft_29 AT %MX21032.29 : BOOL;
	bArm2HorzStn8SlantedLeft_30 AT %MX21032.30 : BOOL;
	bArm2HorzStn8SlantedLeft_31 AT %MX21032.31 : BOOL;

	bArm2HorzStn9SlantedLeft_00 AT %MX21036.0 : BOOL;
	bArm2HorzStn9SlantedLeft_01 AT %MX21036.1 : BOOL;
	bArm2HorzStn9SlantedLeft_02 AT %MX21036.2 : BOOL;
	bArm2HorzStn9SlantedLeft_03 AT %MX21036.3 : BOOL;
	bArm2HorzStn9SlantedLeft_04 AT %MX21036.4 : BOOL;
	bArm2HorzStn9SlantedLeft_05 AT %MX21036.5 : BOOL;
	bArm2HorzStn9SlantedLeft_06 AT %MX21036.6 : BOOL;
	bArm2HorzStn9SlantedLeft_07 AT %MX21036.7 : BOOL;
	bArm2HorzStn9SlantedLeft_08 AT %MX21036.8 : BOOL;
	bArm2HorzStn9SlantedLeft_09 AT %MX21036.9 : BOOL;
	bArm2HorzStn9SlantedLeft_10 AT %MX21036.10 : BOOL;
	bArm2HorzStn9SlantedLeft_11 AT %MX21036.11 : BOOL;
	bArm2HorzStn9SlantedLeft_12 AT %MX21036.12 : BOOL;
	bArm2HorzStn9SlantedLeft_13 AT %MX21036.13 : BOOL;
	bArm2HorzStn9SlantedLeft_14 AT %MX21036.14 : BOOL;
	bArm2HorzStn9SlantedLeft_15 AT %MX21036.15 : BOOL;
	bArm2HorzStn9SlantedLeft_16 AT %MX21036.16 : BOOL;
	bArm2HorzStn9SlantedLeft_17 AT %MX21036.17 : BOOL;
	bArm2HorzStn9SlantedLeft_18 AT %MX21036.18 : BOOL;
	bArm2HorzStn9SlantedLeft_19 AT %MX21036.19 : BOOL;
	bArm2HorzStn9SlantedLeft_20 AT %MX21036.20 : BOOL;
	bArm2HorzStn9SlantedLeft_21 AT %MX21036.21 : BOOL;
	bArm2HorzStn9SlantedLeft_22 AT %MX21036.22 : BOOL;
	bArm2HorzStn9SlantedLeft_23 AT %MX21036.23 : BOOL;
	bArm2HorzStn9SlantedLeft_24 AT %MX21036.24 : BOOL;
	bArm2HorzStn9SlantedLeft_25 AT %MX21036.25 : BOOL;
	bArm2HorzStn9SlantedLeft_26 AT %MX21036.26 : BOOL;
	bArm2HorzStn9SlantedLeft_27 AT %MX21036.27 : BOOL;
	bArm2HorzStn9SlantedLeft_28 AT %MX21036.28 : BOOL;
	bArm2HorzStn9SlantedLeft_29 AT %MX21036.29 : BOOL;
	bArm2HorzStn9SlantedLeft_30 AT %MX21036.30 : BOOL;
	bArm2HorzStn9SlantedLeft_31 AT %MX21036.31 : BOOL;

	bArm2HorzStn10SlantedLeft_00 AT %MX21040.0 : BOOL;
	bArm2HorzStn10SlantedLeft_01 AT %MX21040.1 : BOOL;
	bArm2HorzStn10SlantedLeft_02 AT %MX21040.2 : BOOL;
	bArm2HorzStn10SlantedLeft_03 AT %MX21040.3 : BOOL;
	bArm2HorzStn10SlantedLeft_04 AT %MX21040.4 : BOOL;
	bArm2HorzStn10SlantedLeft_05 AT %MX21040.5 : BOOL;
	bArm2HorzStn10SlantedLeft_06 AT %MX21040.6 : BOOL;
	bArm2HorzStn10SlantedLeft_07 AT %MX21040.7 : BOOL;
	bArm2HorzStn10SlantedLeft_08 AT %MX21040.8 : BOOL;
	bArm2HorzStn10SlantedLeft_09 AT %MX21040.9 : BOOL;
	bArm2HorzStn10SlantedLeft_10 AT %MX21040.10 : BOOL;
	bArm2HorzStn10SlantedLeft_11 AT %MX21040.11 : BOOL;
	bArm2HorzStn10SlantedLeft_12 AT %MX21040.12 : BOOL;
	bArm2HorzStn10SlantedLeft_13 AT %MX21040.13 : BOOL;
	bArm2HorzStn10SlantedLeft_14 AT %MX21040.14 : BOOL;
	bArm2HorzStn10SlantedLeft_15 AT %MX21040.15 : BOOL;
	bArm2HorzStn10SlantedLeft_16 AT %MX21040.16 : BOOL;
	bArm2HorzStn10SlantedLeft_17 AT %MX21040.17 : BOOL;
	bArm2HorzStn10SlantedLeft_18 AT %MX21040.18 : BOOL;
	bArm2HorzStn10SlantedLeft_19 AT %MX21040.19 : BOOL;
	bArm2HorzStn10SlantedLeft_20 AT %MX21040.20 : BOOL;
	bArm2HorzStn10SlantedLeft_21 AT %MX21040.21 : BOOL;
	bArm2HorzStn10SlantedLeft_22 AT %MX21040.22 : BOOL;
	bArm2HorzStn10SlantedLeft_23 AT %MX21040.23 : BOOL;
	bArm2HorzStn10SlantedLeft_24 AT %MX21040.24 : BOOL;
	bArm2HorzStn10SlantedLeft_25 AT %MX21040.25 : BOOL;
	bArm2HorzStn10SlantedLeft_26 AT %MX21040.26 : BOOL;
	bArm2HorzStn10SlantedLeft_27 AT %MX21040.27 : BOOL;
	bArm2HorzStn10SlantedLeft_28 AT %MX21040.28 : BOOL;
	bArm2HorzStn10SlantedLeft_29 AT %MX21040.29 : BOOL;
	bArm2HorzStn10SlantedLeft_30 AT %MX21040.30 : BOOL;
	bArm2HorzStn10SlantedLeft_31 AT %MX21040.31 : BOOL;

	bArm2HorzStn11SlantedLeft_00 AT %MX21044.0 : BOOL;
	bArm2HorzStn11SlantedLeft_01 AT %MX21044.1 : BOOL;
	bArm2HorzStn11SlantedLeft_02 AT %MX21044.2 : BOOL;
	bArm2HorzStn11SlantedLeft_03 AT %MX21044.3 : BOOL;
	bArm2HorzStn11SlantedLeft_04 AT %MX21044.4 : BOOL;
	bArm2HorzStn11SlantedLeft_05 AT %MX21044.5 : BOOL;
	bArm2HorzStn11SlantedLeft_06 AT %MX21044.6 : BOOL;
	bArm2HorzStn11SlantedLeft_07 AT %MX21044.7 : BOOL;
	bArm2HorzStn11SlantedLeft_08 AT %MX21044.8 : BOOL;
	bArm2HorzStn11SlantedLeft_09 AT %MX21044.9 : BOOL;
	bArm2HorzStn11SlantedLeft_10 AT %MX21044.10 : BOOL;
	bArm2HorzStn11SlantedLeft_11 AT %MX21044.11 : BOOL;
	bArm2HorzStn11SlantedLeft_12 AT %MX21044.12 : BOOL;
	bArm2HorzStn11SlantedLeft_13 AT %MX21044.13 : BOOL;
	bArm2HorzStn11SlantedLeft_14 AT %MX21044.14 : BOOL;
	bArm2HorzStn11SlantedLeft_15 AT %MX21044.15 : BOOL;
	bArm2HorzStn11SlantedLeft_16 AT %MX21044.16 : BOOL;
	bArm2HorzStn11SlantedLeft_17 AT %MX21044.17 : BOOL;
	bArm2HorzStn11SlantedLeft_18 AT %MX21044.18 : BOOL;
	bArm2HorzStn11SlantedLeft_19 AT %MX21044.19 : BOOL;
	bArm2HorzStn11SlantedLeft_20 AT %MX21044.20 : BOOL;
	bArm2HorzStn11SlantedLeft_21 AT %MX21044.21 : BOOL;
	bArm2HorzStn11SlantedLeft_22 AT %MX21044.22 : BOOL;
	bArm2HorzStn11SlantedLeft_23 AT %MX21044.23 : BOOL;
	bArm2HorzStn11SlantedLeft_24 AT %MX21044.24 : BOOL;
	bArm2HorzStn11SlantedLeft_25 AT %MX21044.25 : BOOL;
	bArm2HorzStn11SlantedLeft_26 AT %MX21044.26 : BOOL;
	bArm2HorzStn11SlantedLeft_27 AT %MX21044.27 : BOOL;
	bArm2HorzStn11SlantedLeft_28 AT %MX21044.28 : BOOL;
	bArm2HorzStn11SlantedLeft_29 AT %MX21044.29 : BOOL;
	bArm2HorzStn11SlantedLeft_30 AT %MX21044.30 : BOOL;
	bArm2HorzStn11SlantedLeft_31 AT %MX21044.31 : BOOL;

	bArm2HorzStn12SlantedLeft_00 AT %MX21048.0 : BOOL;
	bArm2HorzStn12SlantedLeft_01 AT %MX21048.1 : BOOL;
	bArm2HorzStn12SlantedLeft_02 AT %MX21048.2 : BOOL;
	bArm2HorzStn12SlantedLeft_03 AT %MX21048.3 : BOOL;
	bArm2HorzStn12SlantedLeft_04 AT %MX21048.4 : BOOL;
	bArm2HorzStn12SlantedLeft_05 AT %MX21048.5 : BOOL;
	bArm2HorzStn12SlantedLeft_06 AT %MX21048.6 : BOOL;
	bArm2HorzStn12SlantedLeft_07 AT %MX21048.7 : BOOL;
	bArm2HorzStn12SlantedLeft_08 AT %MX21048.8 : BOOL;
	bArm2HorzStn12SlantedLeft_09 AT %MX21048.9 : BOOL;
	bArm2HorzStn12SlantedLeft_10 AT %MX21048.10 : BOOL;
	bArm2HorzStn12SlantedLeft_11 AT %MX21048.11 : BOOL;
	bArm2HorzStn12SlantedLeft_12 AT %MX21048.12 : BOOL;
	bArm2HorzStn12SlantedLeft_13 AT %MX21048.13 : BOOL;
	bArm2HorzStn12SlantedLeft_14 AT %MX21048.14 : BOOL;
	bArm2HorzStn12SlantedLeft_15 AT %MX21048.15 : BOOL;
	bArm2HorzStn12SlantedLeft_16 AT %MX21048.16 : BOOL;
	bArm2HorzStn12SlantedLeft_17 AT %MX21048.17 : BOOL;
	bArm2HorzStn12SlantedLeft_18 AT %MX21048.18 : BOOL;
	bArm2HorzStn12SlantedLeft_19 AT %MX21048.19 : BOOL;
	bArm2HorzStn12SlantedLeft_20 AT %MX21048.20 : BOOL;
	bArm2HorzStn12SlantedLeft_21 AT %MX21048.21 : BOOL;
	bArm2HorzStn12SlantedLeft_22 AT %MX21048.22 : BOOL;
	bArm2HorzStn12SlantedLeft_23 AT %MX21048.23 : BOOL;
	bArm2HorzStn12SlantedLeft_24 AT %MX21048.24 : BOOL;
	bArm2HorzStn12SlantedLeft_25 AT %MX21048.25 : BOOL;
	bArm2HorzStn12SlantedLeft_26 AT %MX21048.26 : BOOL;
	bArm2HorzStn12SlantedLeft_27 AT %MX21048.27 : BOOL;
	bArm2HorzStn12SlantedLeft_28 AT %MX21048.28 : BOOL;
	bArm2HorzStn12SlantedLeft_29 AT %MX21048.29 : BOOL;
	bArm2HorzStn12SlantedLeft_30 AT %MX21048.30 : BOOL;
	bArm2HorzStn12SlantedLeft_31 AT %MX21048.31 : BOOL;


(*=============================== SlantedRight word ===============================*)
(*====================== SlantedRight BOOL LINK with %MX21100-MX21199 ======================*)

	bArm2HorzStn1SlantedRight_00 AT %MX21104.0 : BOOL;
	bArm2HorzStn1SlantedRight_01 AT %MX21104.1 : BOOL;
	bArm2HorzStn1SlantedRight_02 AT %MX21104.2 : BOOL;
	bArm2HorzStn1SlantedRight_03 AT %MX21104.3 : BOOL;
	bArm2HorzStn1SlantedRight_04 AT %MX21104.4 : BOOL;
	bArm2HorzStn1SlantedRight_05 AT %MX21104.5 : BOOL;
	bArm2HorzStn1SlantedRight_06 AT %MX21104.6 : BOOL;
	bArm2HorzStn1SlantedRight_07 AT %MX21104.7 : BOOL;
	bArm2HorzStn1SlantedRight_08 AT %MX21104.8 : BOOL;
	bArm2HorzStn1SlantedRight_09 AT %MX21104.9 : BOOL;
	bArm2HorzStn1SlantedRight_10 AT %MX21104.10 : BOOL;
	bArm2HorzStn1SlantedRight_11 AT %MX21104.11 : BOOL;
	bArm2HorzStn1SlantedRight_12 AT %MX21104.12 : BOOL;
	bArm2HorzStn1SlantedRight_13 AT %MX21104.13 : BOOL;
	bArm2HorzStn1SlantedRight_14 AT %MX21104.14 : BOOL;
	bArm2HorzStn1SlantedRight_15 AT %MX21104.15 : BOOL;
	bArm2HorzStn1SlantedRight_16 AT %MX21104.16 : BOOL;
	bArm2HorzStn1SlantedRight_17 AT %MX21104.17 : BOOL;
	bArm2HorzStn1SlantedRight_18 AT %MX21104.18 : BOOL;
	bArm2HorzStn1SlantedRight_19 AT %MX21104.19 : BOOL;
	bArm2HorzStn1SlantedRight_20 AT %MX21104.20 : BOOL;
	bArm2HorzStn1SlantedRight_21 AT %MX21104.21 : BOOL;
	bArm2HorzStn1SlantedRight_22 AT %MX21104.22 : BOOL;
	bArm2HorzStn1SlantedRight_23 AT %MX21104.23 : BOOL;
	bArm2HorzStn1SlantedRight_24 AT %MX21104.24 : BOOL;
	bArm2HorzStn1SlantedRight_25 AT %MX21104.25 : BOOL;
	bArm2HorzStn1SlantedRight_26 AT %MX21104.26 : BOOL;
	bArm2HorzStn1SlantedRight_27 AT %MX21104.27 : BOOL;
	bArm2HorzStn1SlantedRight_28 AT %MX21104.28 : BOOL;
	bArm2HorzStn1SlantedRight_29 AT %MX21104.29 : BOOL;
	bArm2HorzStn1SlantedRight_30 AT %MX21104.30 : BOOL;
	bArm2HorzStn1SlantedRight_31 AT %MX21104.31 : BOOL;

	bArm2HorzStn2SlantedRight_00 AT %MX21108.0 : BOOL;
	bArm2HorzStn2SlantedRight_01 AT %MX21108.1 : BOOL;
	bArm2HorzStn2SlantedRight_02 AT %MX21108.2 : BOOL;
	bArm2HorzStn2SlantedRight_03 AT %MX21108.3 : BOOL;
	bArm2HorzStn2SlantedRight_04 AT %MX21108.4 : BOOL;
	bArm2HorzStn2SlantedRight_05 AT %MX21108.5 : BOOL;
	bArm2HorzStn2SlantedRight_06 AT %MX21108.6 : BOOL;
	bArm2HorzStn2SlantedRight_07 AT %MX21108.7 : BOOL;
	bArm2HorzStn2SlantedRight_08 AT %MX21108.8 : BOOL;
	bArm2HorzStn2SlantedRight_09 AT %MX21108.9 : BOOL;
	bArm2HorzStn2SlantedRight_10 AT %MX21108.10 : BOOL;
	bArm2HorzStn2SlantedRight_11 AT %MX21108.11 : BOOL;
	bArm2HorzStn2SlantedRight_12 AT %MX21108.12 : BOOL;
	bArm2HorzStn2SlantedRight_13 AT %MX21108.13 : BOOL;
	bArm2HorzStn2SlantedRight_14 AT %MX21108.14 : BOOL;
	bArm2HorzStn2SlantedRight_15 AT %MX21108.15 : BOOL;
	bArm2HorzStn2SlantedRight_16 AT %MX21108.16 : BOOL;
	bArm2HorzStn2SlantedRight_17 AT %MX21108.17 : BOOL;
	bArm2HorzStn2SlantedRight_18 AT %MX21108.18 : BOOL;
	bArm2HorzStn2SlantedRight_19 AT %MX21108.19 : BOOL;
	bArm2HorzStn2SlantedRight_20 AT %MX21108.20 : BOOL;
	bArm2HorzStn2SlantedRight_21 AT %MX21108.21 : BOOL;
	bArm2HorzStn2SlantedRight_22 AT %MX21108.22 : BOOL;
	bArm2HorzStn2SlantedRight_23 AT %MX21108.23 : BOOL;
	bArm2HorzStn2SlantedRight_24 AT %MX21108.24 : BOOL;
	bArm2HorzStn2SlantedRight_25 AT %MX21108.25 : BOOL;
	bArm2HorzStn2SlantedRight_26 AT %MX21108.26 : BOOL;
	bArm2HorzStn2SlantedRight_27 AT %MX21108.27 : BOOL;
	bArm2HorzStn2SlantedRight_28 AT %MX21108.28 : BOOL;
	bArm2HorzStn2SlantedRight_29 AT %MX21108.29 : BOOL;
	bArm2HorzStn2SlantedRight_30 AT %MX21108.30 : BOOL;
	bArm2HorzStn2SlantedRight_31 AT %MX21108.31 : BOOL;

	bArm2HorzStn3SlantedRight_00 AT %MX21112.0 : BOOL;
	bArm2HorzStn3SlantedRight_01 AT %MX21112.1 : BOOL;
	bArm2HorzStn3SlantedRight_02 AT %MX21112.2 : BOOL;
	bArm2HorzStn3SlantedRight_03 AT %MX21112.3 : BOOL;
	bArm2HorzStn3SlantedRight_04 AT %MX21112.4 : BOOL;
	bArm2HorzStn3SlantedRight_05 AT %MX21112.5 : BOOL;
	bArm2HorzStn3SlantedRight_06 AT %MX21112.6 : BOOL;
	bArm2HorzStn3SlantedRight_07 AT %MX21112.7 : BOOL;
	bArm2HorzStn3SlantedRight_08 AT %MX21112.8 : BOOL;
	bArm2HorzStn3SlantedRight_09 AT %MX21112.9 : BOOL;
	bArm2HorzStn3SlantedRight_10 AT %MX21112.10 : BOOL;
	bArm2HorzStn3SlantedRight_11 AT %MX21112.11 : BOOL;
	bArm2HorzStn3SlantedRight_12 AT %MX21112.12 : BOOL;
	bArm2HorzStn3SlantedRight_13 AT %MX21112.13 : BOOL;
	bArm2HorzStn3SlantedRight_14 AT %MX21112.14 : BOOL;
	bArm2HorzStn3SlantedRight_15 AT %MX21112.15 : BOOL;
	bArm2HorzStn3SlantedRight_16 AT %MX21112.16 : BOOL;
	bArm2HorzStn3SlantedRight_17 AT %MX21112.17 : BOOL;
	bArm2HorzStn3SlantedRight_18 AT %MX21112.18 : BOOL;
	bArm2HorzStn3SlantedRight_19 AT %MX21112.19 : BOOL;
	bArm2HorzStn3SlantedRight_20 AT %MX21112.20 : BOOL;
	bArm2HorzStn3SlantedRight_21 AT %MX21112.21 : BOOL;
	bArm2HorzStn3SlantedRight_22 AT %MX21112.22 : BOOL;
	bArm2HorzStn3SlantedRight_23 AT %MX21112.23 : BOOL;
	bArm2HorzStn3SlantedRight_24 AT %MX21112.24 : BOOL;
	bArm2HorzStn3SlantedRight_25 AT %MX21112.25 : BOOL;
	bArm2HorzStn3SlantedRight_26 AT %MX21112.26 : BOOL;
	bArm2HorzStn3SlantedRight_27 AT %MX21112.27 : BOOL;
	bArm2HorzStn3SlantedRight_28 AT %MX21112.28 : BOOL;
	bArm2HorzStn3SlantedRight_29 AT %MX21112.29 : BOOL;
	bArm2HorzStn3SlantedRight_30 AT %MX21112.30 : BOOL;
	bArm2HorzStn3SlantedRight_31 AT %MX21112.31 : BOOL;

	bArm2HorzStn4SlantedRight_00 AT %MX21116.0 : BOOL;
	bArm2HorzStn4SlantedRight_01 AT %MX21116.1 : BOOL;
	bArm2HorzStn4SlantedRight_02 AT %MX21116.2 : BOOL;
	bArm2HorzStn4SlantedRight_03 AT %MX21116.3 : BOOL;
	bArm2HorzStn4SlantedRight_04 AT %MX21116.4 : BOOL;
	bArm2HorzStn4SlantedRight_05 AT %MX21116.5 : BOOL;
	bArm2HorzStn4SlantedRight_06 AT %MX21116.6 : BOOL;
	bArm2HorzStn4SlantedRight_07 AT %MX21116.7 : BOOL;
	bArm2HorzStn4SlantedRight_08 AT %MX21116.8 : BOOL;
	bArm2HorzStn4SlantedRight_09 AT %MX21116.9 : BOOL;
	bArm2HorzStn4SlantedRight_10 AT %MX21116.10 : BOOL;
	bArm2HorzStn4SlantedRight_11 AT %MX21116.11 : BOOL;
	bArm2HorzStn4SlantedRight_12 AT %MX21116.12 : BOOL;
	bArm2HorzStn4SlantedRight_13 AT %MX21116.13 : BOOL;
	bArm2HorzStn4SlantedRight_14 AT %MX21116.14 : BOOL;
	bArm2HorzStn4SlantedRight_15 AT %MX21116.15 : BOOL;
	bArm2HorzStn4SlantedRight_16 AT %MX21116.16 : BOOL;
	bArm2HorzStn4SlantedRight_17 AT %MX21116.17 : BOOL;
	bArm2HorzStn4SlantedRight_18 AT %MX21116.18 : BOOL;
	bArm2HorzStn4SlantedRight_19 AT %MX21116.19 : BOOL;
	bArm2HorzStn4SlantedRight_20 AT %MX21116.20 : BOOL;
	bArm2HorzStn4SlantedRight_21 AT %MX21116.21 : BOOL;
	bArm2HorzStn4SlantedRight_22 AT %MX21116.22 : BOOL;
	bArm2HorzStn4SlantedRight_23 AT %MX21116.23 : BOOL;
	bArm2HorzStn4SlantedRight_24 AT %MX21116.24 : BOOL;
	bArm2HorzStn4SlantedRight_25 AT %MX21116.25 : BOOL;
	bArm2HorzStn4SlantedRight_26 AT %MX21116.26 : BOOL;
	bArm2HorzStn4SlantedRight_27 AT %MX21116.27 : BOOL;
	bArm2HorzStn4SlantedRight_28 AT %MX21116.28 : BOOL;
	bArm2HorzStn4SlantedRight_29 AT %MX21116.29 : BOOL;
	bArm2HorzStn4SlantedRight_30 AT %MX21116.30 : BOOL;
	bArm2HorzStn4SlantedRight_31 AT %MX21116.31 : BOOL;

	bArm2HorzStn5SlantedRight_00 AT %MX21120.0 : BOOL;
	bArm2HorzStn5SlantedRight_01 AT %MX21120.1 : BOOL;
	bArm2HorzStn5SlantedRight_02 AT %MX21120.2 : BOOL;
	bArm2HorzStn5SlantedRight_03 AT %MX21120.3 : BOOL;
	bArm2HorzStn5SlantedRight_04 AT %MX21120.4 : BOOL;
	bArm2HorzStn5SlantedRight_05 AT %MX21120.5 : BOOL;
	bArm2HorzStn5SlantedRight_06 AT %MX21120.6 : BOOL;
	bArm2HorzStn5SlantedRight_07 AT %MX21120.7 : BOOL;
	bArm2HorzStn5SlantedRight_08 AT %MX21120.8 : BOOL;
	bArm2HorzStn5SlantedRight_09 AT %MX21120.9 : BOOL;
	bArm2HorzStn5SlantedRight_10 AT %MX21120.10 : BOOL;
	bArm2HorzStn5SlantedRight_11 AT %MX21120.11 : BOOL;
	bArm2HorzStn5SlantedRight_12 AT %MX21120.12 : BOOL;
	bArm2HorzStn5SlantedRight_13 AT %MX21120.13 : BOOL;
	bArm2HorzStn5SlantedRight_14 AT %MX21120.14 : BOOL;
	bArm2HorzStn5SlantedRight_15 AT %MX21120.15 : BOOL;
	bArm2HorzStn5SlantedRight_16 AT %MX21120.16 : BOOL;
	bArm2HorzStn5SlantedRight_17 AT %MX21120.17 : BOOL;
	bArm2HorzStn5SlantedRight_18 AT %MX21120.18 : BOOL;
	bArm2HorzStn5SlantedRight_19 AT %MX21120.19 : BOOL;
	bArm2HorzStn5SlantedRight_20 AT %MX21120.20 : BOOL;
	bArm2HorzStn5SlantedRight_21 AT %MX21120.21 : BOOL;
	bArm2HorzStn5SlantedRight_22 AT %MX21120.22 : BOOL;
	bArm2HorzStn5SlantedRight_23 AT %MX21120.23 : BOOL;
	bArm2HorzStn5SlantedRight_24 AT %MX21120.24 : BOOL;
	bArm2HorzStn5SlantedRight_25 AT %MX21120.25 : BOOL;
	bArm2HorzStn5SlantedRight_26 AT %MX21120.26 : BOOL;
	bArm2HorzStn5SlantedRight_27 AT %MX21120.27 : BOOL;
	bArm2HorzStn5SlantedRight_28 AT %MX21120.28 : BOOL;
	bArm2HorzStn5SlantedRight_29 AT %MX21120.29 : BOOL;
	bArm2HorzStn5SlantedRight_30 AT %MX21120.30 : BOOL;
	bArm2HorzStn5SlantedRight_31 AT %MX21120.31 : BOOL;

	bArm2HorzStn6SlantedRight_00 AT %MX21124.0 : BOOL;
	bArm2HorzStn6SlantedRight_01 AT %MX21124.1 : BOOL;
	bArm2HorzStn6SlantedRight_02 AT %MX21124.2 : BOOL;
	bArm2HorzStn6SlantedRight_03 AT %MX21124.3 : BOOL;
	bArm2HorzStn6SlantedRight_04 AT %MX21124.4 : BOOL;
	bArm2HorzStn6SlantedRight_05 AT %MX21124.5 : BOOL;
	bArm2HorzStn6SlantedRight_06 AT %MX21124.6 : BOOL;
	bArm2HorzStn6SlantedRight_07 AT %MX21124.7 : BOOL;
	bArm2HorzStn6SlantedRight_08 AT %MX21124.8 : BOOL;
	bArm2HorzStn6SlantedRight_09 AT %MX21124.9 : BOOL;
	bArm2HorzStn6SlantedRight_10 AT %MX21124.10 : BOOL;
	bArm2HorzStn6SlantedRight_11 AT %MX21124.11 : BOOL;
	bArm2HorzStn6SlantedRight_12 AT %MX21124.12 : BOOL;
	bArm2HorzStn6SlantedRight_13 AT %MX21124.13 : BOOL;
	bArm2HorzStn6SlantedRight_14 AT %MX21124.14 : BOOL;
	bArm2HorzStn6SlantedRight_15 AT %MX21124.15 : BOOL;
	bArm2HorzStn6SlantedRight_16 AT %MX21124.16 : BOOL;
	bArm2HorzStn6SlantedRight_17 AT %MX21124.17 : BOOL;
	bArm2HorzStn6SlantedRight_18 AT %MX21124.18 : BOOL;
	bArm2HorzStn6SlantedRight_19 AT %MX21124.19 : BOOL;
	bArm2HorzStn6SlantedRight_20 AT %MX21124.20 : BOOL;
	bArm2HorzStn6SlantedRight_21 AT %MX21124.21 : BOOL;
	bArm2HorzStn6SlantedRight_22 AT %MX21124.22 : BOOL;
	bArm2HorzStn6SlantedRight_23 AT %MX21124.23 : BOOL;
	bArm2HorzStn6SlantedRight_24 AT %MX21124.24 : BOOL;
	bArm2HorzStn6SlantedRight_25 AT %MX21124.25 : BOOL;
	bArm2HorzStn6SlantedRight_26 AT %MX21124.26 : BOOL;
	bArm2HorzStn6SlantedRight_27 AT %MX21124.27 : BOOL;
	bArm2HorzStn6SlantedRight_28 AT %MX21124.28 : BOOL;
	bArm2HorzStn6SlantedRight_29 AT %MX21124.29 : BOOL;
	bArm2HorzStn6SlantedRight_30 AT %MX21124.30 : BOOL;
	bArm2HorzStn6SlantedRight_31 AT %MX21124.31 : BOOL;

	bArm2HorzStn7SlantedRight_00 AT %MX21128.0 : BOOL;
	bArm2HorzStn7SlantedRight_01 AT %MX21128.1 : BOOL;
	bArm2HorzStn7SlantedRight_02 AT %MX21128.2 : BOOL;
	bArm2HorzStn7SlantedRight_03 AT %MX21128.3 : BOOL;
	bArm2HorzStn7SlantedRight_04 AT %MX21128.4 : BOOL;
	bArm2HorzStn7SlantedRight_05 AT %MX21128.5 : BOOL;
	bArm2HorzStn7SlantedRight_06 AT %MX21128.6 : BOOL;
	bArm2HorzStn7SlantedRight_07 AT %MX21128.7 : BOOL;
	bArm2HorzStn7SlantedRight_08 AT %MX21128.8 : BOOL;
	bArm2HorzStn7SlantedRight_09 AT %MX21128.9 : BOOL;
	bArm2HorzStn7SlantedRight_10 AT %MX21128.10 : BOOL;
	bArm2HorzStn7SlantedRight_11 AT %MX21128.11 : BOOL;
	bArm2HorzStn7SlantedRight_12 AT %MX21128.12 : BOOL;
	bArm2HorzStn7SlantedRight_13 AT %MX21128.13 : BOOL;
	bArm2HorzStn7SlantedRight_14 AT %MX21128.14 : BOOL;
	bArm2HorzStn7SlantedRight_15 AT %MX21128.15 : BOOL;
	bArm2HorzStn7SlantedRight_16 AT %MX21128.16 : BOOL;
	bArm2HorzStn7SlantedRight_17 AT %MX21128.17 : BOOL;
	bArm2HorzStn7SlantedRight_18 AT %MX21128.18 : BOOL;
	bArm2HorzStn7SlantedRight_19 AT %MX21128.19 : BOOL;
	bArm2HorzStn7SlantedRight_20 AT %MX21128.20 : BOOL;
	bArm2HorzStn7SlantedRight_21 AT %MX21128.21 : BOOL;
	bArm2HorzStn7SlantedRight_22 AT %MX21128.22 : BOOL;
	bArm2HorzStn7SlantedRight_23 AT %MX21128.23 : BOOL;
	bArm2HorzStn7SlantedRight_24 AT %MX21128.24 : BOOL;
	bArm2HorzStn7SlantedRight_25 AT %MX21128.25 : BOOL;
	bArm2HorzStn7SlantedRight_26 AT %MX21128.26 : BOOL;
	bArm2HorzStn7SlantedRight_27 AT %MX21128.27 : BOOL;
	bArm2HorzStn7SlantedRight_28 AT %MX21128.28 : BOOL;
	bArm2HorzStn7SlantedRight_29 AT %MX21128.29 : BOOL;
	bArm2HorzStn7SlantedRight_30 AT %MX21128.30 : BOOL;
	bArm2HorzStn7SlantedRight_31 AT %MX21128.31 : BOOL;

	bArm2HorzStn8SlantedRight_00 AT %MX21132.0 : BOOL;
	bArm2HorzStn8SlantedRight_01 AT %MX21132.1 : BOOL;
	bArm2HorzStn8SlantedRight_02 AT %MX21132.2 : BOOL;
	bArm2HorzStn8SlantedRight_03 AT %MX21132.3 : BOOL;
	bArm2HorzStn8SlantedRight_04 AT %MX21132.4 : BOOL;
	bArm2HorzStn8SlantedRight_05 AT %MX21132.5 : BOOL;
	bArm2HorzStn8SlantedRight_06 AT %MX21132.6 : BOOL;
	bArm2HorzStn8SlantedRight_07 AT %MX21132.7 : BOOL;
	bArm2HorzStn8SlantedRight_08 AT %MX21132.8 : BOOL;
	bArm2HorzStn8SlantedRight_09 AT %MX21132.9 : BOOL;
	bArm2HorzStn8SlantedRight_10 AT %MX21132.10 : BOOL;
	bArm2HorzStn8SlantedRight_11 AT %MX21132.11 : BOOL;
	bArm2HorzStn8SlantedRight_12 AT %MX21132.12 : BOOL;
	bArm2HorzStn8SlantedRight_13 AT %MX21132.13 : BOOL;
	bArm2HorzStn8SlantedRight_14 AT %MX21132.14 : BOOL;
	bArm2HorzStn8SlantedRight_15 AT %MX21132.15 : BOOL;
	bArm2HorzStn8SlantedRight_16 AT %MX21132.16 : BOOL;
	bArm2HorzStn8SlantedRight_17 AT %MX21132.17 : BOOL;
	bArm2HorzStn8SlantedRight_18 AT %MX21132.18 : BOOL;
	bArm2HorzStn8SlantedRight_19 AT %MX21132.19 : BOOL;
	bArm2HorzStn8SlantedRight_20 AT %MX21132.20 : BOOL;
	bArm2HorzStn8SlantedRight_21 AT %MX21132.21 : BOOL;
	bArm2HorzStn8SlantedRight_22 AT %MX21132.22 : BOOL;
	bArm2HorzStn8SlantedRight_23 AT %MX21132.23 : BOOL;
	bArm2HorzStn8SlantedRight_24 AT %MX21132.24 : BOOL;
	bArm2HorzStn8SlantedRight_25 AT %MX21132.25 : BOOL;
	bArm2HorzStn8SlantedRight_26 AT %MX21132.26 : BOOL;
	bArm2HorzStn8SlantedRight_27 AT %MX21132.27 : BOOL;
	bArm2HorzStn8SlantedRight_28 AT %MX21132.28 : BOOL;
	bArm2HorzStn8SlantedRight_29 AT %MX21132.29 : BOOL;
	bArm2HorzStn8SlantedRight_30 AT %MX21132.30 : BOOL;
	bArm2HorzStn8SlantedRight_31 AT %MX21132.31 : BOOL;

	bArm2HorzStn9SlantedRight_00 AT %MX21136.0 : BOOL;
	bArm2HorzStn9SlantedRight_01 AT %MX21136.1 : BOOL;
	bArm2HorzStn9SlantedRight_02 AT %MX21136.2 : BOOL;
	bArm2HorzStn9SlantedRight_03 AT %MX21136.3 : BOOL;
	bArm2HorzStn9SlantedRight_04 AT %MX21136.4 : BOOL;
	bArm2HorzStn9SlantedRight_05 AT %MX21136.5 : BOOL;
	bArm2HorzStn9SlantedRight_06 AT %MX21136.6 : BOOL;
	bArm2HorzStn9SlantedRight_07 AT %MX21136.7 : BOOL;
	bArm2HorzStn9SlantedRight_08 AT %MX21136.8 : BOOL;
	bArm2HorzStn9SlantedRight_09 AT %MX21136.9 : BOOL;
	bArm2HorzStn9SlantedRight_10 AT %MX21136.10 : BOOL;
	bArm2HorzStn9SlantedRight_11 AT %MX21136.11 : BOOL;
	bArm2HorzStn9SlantedRight_12 AT %MX21136.12 : BOOL;
	bArm2HorzStn9SlantedRight_13 AT %MX21136.13 : BOOL;
	bArm2HorzStn9SlantedRight_14 AT %MX21136.14 : BOOL;
	bArm2HorzStn9SlantedRight_15 AT %MX21136.15 : BOOL;
	bArm2HorzStn9SlantedRight_16 AT %MX21136.16 : BOOL;
	bArm2HorzStn9SlantedRight_17 AT %MX21136.17 : BOOL;
	bArm2HorzStn9SlantedRight_18 AT %MX21136.18 : BOOL;
	bArm2HorzStn9SlantedRight_19 AT %MX21136.19 : BOOL;
	bArm2HorzStn9SlantedRight_20 AT %MX21136.20 : BOOL;
	bArm2HorzStn9SlantedRight_21 AT %MX21136.21 : BOOL;
	bArm2HorzStn9SlantedRight_22 AT %MX21136.22 : BOOL;
	bArm2HorzStn9SlantedRight_23 AT %MX21136.23 : BOOL;
	bArm2HorzStn9SlantedRight_24 AT %MX21136.24 : BOOL;
	bArm2HorzStn9SlantedRight_25 AT %MX21136.25 : BOOL;
	bArm2HorzStn9SlantedRight_26 AT %MX21136.26 : BOOL;
	bArm2HorzStn9SlantedRight_27 AT %MX21136.27 : BOOL;
	bArm2HorzStn9SlantedRight_28 AT %MX21136.28 : BOOL;
	bArm2HorzStn9SlantedRight_29 AT %MX21136.29 : BOOL;
	bArm2HorzStn9SlantedRight_30 AT %MX21136.30 : BOOL;
	bArm2HorzStn9SlantedRight_31 AT %MX21136.31 : BOOL;

	bArm2HorzStn10SlantedRight_00 AT %MX21140.0 : BOOL;
	bArm2HorzStn10SlantedRight_01 AT %MX21140.1 : BOOL;
	bArm2HorzStn10SlantedRight_02 AT %MX21140.2 : BOOL;
	bArm2HorzStn10SlantedRight_03 AT %MX21140.3 : BOOL;
	bArm2HorzStn10SlantedRight_04 AT %MX21140.4 : BOOL;
	bArm2HorzStn10SlantedRight_05 AT %MX21140.5 : BOOL;
	bArm2HorzStn10SlantedRight_06 AT %MX21140.6 : BOOL;
	bArm2HorzStn10SlantedRight_07 AT %MX21140.7 : BOOL;
	bArm2HorzStn10SlantedRight_08 AT %MX21140.8 : BOOL;
	bArm2HorzStn10SlantedRight_09 AT %MX21140.9 : BOOL;
	bArm2HorzStn10SlantedRight_10 AT %MX21140.10 : BOOL;
	bArm2HorzStn10SlantedRight_11 AT %MX21140.11 : BOOL;
	bArm2HorzStn10SlantedRight_12 AT %MX21140.12 : BOOL;
	bArm2HorzStn10SlantedRight_13 AT %MX21140.13 : BOOL;
	bArm2HorzStn10SlantedRight_14 AT %MX21140.14 : BOOL;
	bArm2HorzStn10SlantedRight_15 AT %MX21140.15 : BOOL;
	bArm2HorzStn10SlantedRight_16 AT %MX21140.16 : BOOL;
	bArm2HorzStn10SlantedRight_17 AT %MX21140.17 : BOOL;
	bArm2HorzStn10SlantedRight_18 AT %MX21140.18 : BOOL;
	bArm2HorzStn10SlantedRight_19 AT %MX21140.19 : BOOL;
	bArm2HorzStn10SlantedRight_20 AT %MX21140.20 : BOOL;
	bArm2HorzStn10SlantedRight_21 AT %MX21140.21 : BOOL;
	bArm2HorzStn10SlantedRight_22 AT %MX21140.22 : BOOL;
	bArm2HorzStn10SlantedRight_23 AT %MX21140.23 : BOOL;
	bArm2HorzStn10SlantedRight_24 AT %MX21140.24 : BOOL;
	bArm2HorzStn10SlantedRight_25 AT %MX21140.25 : BOOL;
	bArm2HorzStn10SlantedRight_26 AT %MX21140.26 : BOOL;
	bArm2HorzStn10SlantedRight_27 AT %MX21140.27 : BOOL;
	bArm2HorzStn10SlantedRight_28 AT %MX21140.28 : BOOL;
	bArm2HorzStn10SlantedRight_29 AT %MX21140.29 : BOOL;
	bArm2HorzStn10SlantedRight_30 AT %MX21140.30 : BOOL;
	bArm2HorzStn10SlantedRight_31 AT %MX21140.31 : BOOL;

	bArm2HorzStn11SlantedRight_00 AT %MX21144.0 : BOOL;
	bArm2HorzStn11SlantedRight_01 AT %MX21144.1 : BOOL;
	bArm2HorzStn11SlantedRight_02 AT %MX21144.2 : BOOL;
	bArm2HorzStn11SlantedRight_03 AT %MX21144.3 : BOOL;
	bArm2HorzStn11SlantedRight_04 AT %MX21144.4 : BOOL;
	bArm2HorzStn11SlantedRight_05 AT %MX21144.5 : BOOL;
	bArm2HorzStn11SlantedRight_06 AT %MX21144.6 : BOOL;
	bArm2HorzStn11SlantedRight_07 AT %MX21144.7 : BOOL;
	bArm2HorzStn11SlantedRight_08 AT %MX21144.8 : BOOL;
	bArm2HorzStn11SlantedRight_09 AT %MX21144.9 : BOOL;
	bArm2HorzStn11SlantedRight_10 AT %MX21144.10 : BOOL;
	bArm2HorzStn11SlantedRight_11 AT %MX21144.11 : BOOL;
	bArm2HorzStn11SlantedRight_12 AT %MX21144.12 : BOOL;
	bArm2HorzStn11SlantedRight_13 AT %MX21144.13 : BOOL;
	bArm2HorzStn11SlantedRight_14 AT %MX21144.14 : BOOL;
	bArm2HorzStn11SlantedRight_15 AT %MX21144.15 : BOOL;
	bArm2HorzStn11SlantedRight_16 AT %MX21144.16 : BOOL;
	bArm2HorzStn11SlantedRight_17 AT %MX21144.17 : BOOL;
	bArm2HorzStn11SlantedRight_18 AT %MX21144.18 : BOOL;
	bArm2HorzStn11SlantedRight_19 AT %MX21144.19 : BOOL;
	bArm2HorzStn11SlantedRight_20 AT %MX21144.20 : BOOL;
	bArm2HorzStn11SlantedRight_21 AT %MX21144.21 : BOOL;
	bArm2HorzStn11SlantedRight_22 AT %MX21144.22 : BOOL;
	bArm2HorzStn11SlantedRight_23 AT %MX21144.23 : BOOL;
	bArm2HorzStn11SlantedRight_24 AT %MX21144.24 : BOOL;
	bArm2HorzStn11SlantedRight_25 AT %MX21144.25 : BOOL;
	bArm2HorzStn11SlantedRight_26 AT %MX21144.26 : BOOL;
	bArm2HorzStn11SlantedRight_27 AT %MX21144.27 : BOOL;
	bArm2HorzStn11SlantedRight_28 AT %MX21144.28 : BOOL;
	bArm2HorzStn11SlantedRight_29 AT %MX21144.29 : BOOL;
	bArm2HorzStn11SlantedRight_30 AT %MX21144.30 : BOOL;
	bArm2HorzStn11SlantedRight_31 AT %MX21144.31 : BOOL;

	bArm2HorzStn12SlantedRight_00 AT %MX21148.0 : BOOL;
	bArm2HorzStn12SlantedRight_01 AT %MX21148.1 : BOOL;
	bArm2HorzStn12SlantedRight_02 AT %MX21148.2 : BOOL;
	bArm2HorzStn12SlantedRight_03 AT %MX21148.3 : BOOL;
	bArm2HorzStn12SlantedRight_04 AT %MX21148.4 : BOOL;
	bArm2HorzStn12SlantedRight_05 AT %MX21148.5 : BOOL;
	bArm2HorzStn12SlantedRight_06 AT %MX21148.6 : BOOL;
	bArm2HorzStn12SlantedRight_07 AT %MX21148.7 : BOOL;
	bArm2HorzStn12SlantedRight_08 AT %MX21148.8 : BOOL;
	bArm2HorzStn12SlantedRight_09 AT %MX21148.9 : BOOL;
	bArm2HorzStn12SlantedRight_10 AT %MX21148.10 : BOOL;
	bArm2HorzStn12SlantedRight_11 AT %MX21148.11 : BOOL;
	bArm2HorzStn12SlantedRight_12 AT %MX21148.12 : BOOL;
	bArm2HorzStn12SlantedRight_13 AT %MX21148.13 : BOOL;
	bArm2HorzStn12SlantedRight_14 AT %MX21148.14 : BOOL;
	bArm2HorzStn12SlantedRight_15 AT %MX21148.15 : BOOL;
	bArm2HorzStn12SlantedRight_16 AT %MX21148.16 : BOOL;
	bArm2HorzStn12SlantedRight_17 AT %MX21148.17 : BOOL;
	bArm2HorzStn12SlantedRight_18 AT %MX21148.18 : BOOL;
	bArm2HorzStn12SlantedRight_19 AT %MX21148.19 : BOOL;
	bArm2HorzStn12SlantedRight_20 AT %MX21148.20 : BOOL;
	bArm2HorzStn12SlantedRight_21 AT %MX21148.21 : BOOL;
	bArm2HorzStn12SlantedRight_22 AT %MX21148.22 : BOOL;
	bArm2HorzStn12SlantedRight_23 AT %MX21148.23 : BOOL;
	bArm2HorzStn12SlantedRight_24 AT %MX21148.24 : BOOL;
	bArm2HorzStn12SlantedRight_25 AT %MX21148.25 : BOOL;
	bArm2HorzStn12SlantedRight_26 AT %MX21148.26 : BOOL;
	bArm2HorzStn12SlantedRight_27 AT %MX21148.27 : BOOL;
	bArm2HorzStn12SlantedRight_28 AT %MX21148.28 : BOOL;
	bArm2HorzStn12SlantedRight_29 AT %MX21148.29 : BOOL;
	bArm2HorzStn12SlantedRight_30 AT %MX21148.30 : BOOL;
	bArm2HorzStn12SlantedRight_31 AT %MX21148.31 : BOOL;

(*=============================== Hook word ===============================*)
(*====================== Hook BOOL LINK with %MX21200-MX21299 ======================*)

	bArm2HorzLD1Hook_00 AT %MX21252.0 : BOOL;
	bArm2HorzLD1Hook_01 AT %MX21252.1 : BOOL;
	bArm2HorzLD1Hook_02 AT %MX21252.2 : BOOL;
	bArm2HorzLD1Hook_03 AT %MX21252.3 : BOOL;
	bArm2HorzLD1Hook_04 AT %MX21252.4 : BOOL;
	bArm2HorzLD1Hook_05 AT %MX21252.5 : BOOL;
	bArm2HorzLD1Hook_06 AT %MX21252.6 : BOOL;
	bArm2HorzLD1Hook_07 AT %MX21252.7 : BOOL;
	bArm2HorzLD1Hook_08 AT %MX21252.8 : BOOL;
	bArm2HorzLD1Hook_09 AT %MX21252.9 : BOOL;
	bArm2HorzLD1Hook_10 AT %MX21252.10 : BOOL;
	bArm2HorzLD1Hook_11 AT %MX21252.11 : BOOL;
	bArm2HorzLD1Hook_12 AT %MX21252.12 : BOOL;
	bArm2HorzLD1Hook_13 AT %MX21252.13 : BOOL;
	bArm2HorzLD1Hook_14 AT %MX21252.14 : BOOL;
	bArm2HorzLD1Hook_15 AT %MX21252.15 : BOOL;
	bArm2HorzLD1Hook_16 AT %MX21252.16 : BOOL;
	bArm2HorzLD1Hook_17 AT %MX21252.17 : BOOL;
	bArm2HorzLD1Hook_18 AT %MX21252.18 : BOOL;
	bArm2HorzLD1Hook_19 AT %MX21252.19 : BOOL;
	bArm2HorzLD1Hook_20 AT %MX21252.20 : BOOL;
	bArm2HorzLD1Hook_21 AT %MX21252.21 : BOOL;
	bArm2HorzLD1Hook_22 AT %MX21252.22 : BOOL;
	bArm2HorzLD1Hook_23 AT %MX21252.23 : BOOL;
	bArm2HorzLD1Hook_24 AT %MX21252.24 : BOOL;
	bArm2HorzLD1Hook_25 AT %MX21252.25 : BOOL;
	bArm2HorzLD1Hook_26 AT %MX21252.26 : BOOL;
	bArm2HorzLD1Hook_27 AT %MX21252.27 : BOOL;
	bArm2HorzLD1Hook_28 AT %MX21252.28 : BOOL;
	bArm2HorzLD1Hook_29 AT %MX21252.29 : BOOL;
	bArm2HorzLD1Hook_30 AT %MX21252.30 : BOOL;
	bArm2HorzLD1Hook_31 AT %MX21252.31 : BOOL;

	bArm2HorzULD1Hook_00 AT %MX21256.0 : BOOL;
	bArm2HorzULD1Hook_01 AT %MX21256.1 : BOOL;
	bArm2HorzULD1Hook_02 AT %MX21256.2 : BOOL;
	bArm2HorzULD1Hook_03 AT %MX21256.3 : BOOL;
	bArm2HorzULD1Hook_04 AT %MX21256.4 : BOOL;
	bArm2HorzULD1Hook_05 AT %MX21256.5 : BOOL;
	bArm2HorzULD1Hook_06 AT %MX21256.6 : BOOL;
	bArm2HorzULD1Hook_07 AT %MX21256.7 : BOOL;
	bArm2HorzULD1Hook_08 AT %MX21256.8 : BOOL;
	bArm2HorzULD1Hook_09 AT %MX21256.9 : BOOL;
	bArm2HorzULD1Hook_10 AT %MX21256.10 : BOOL;
	bArm2HorzULD1Hook_11 AT %MX21256.11 : BOOL;
	bArm2HorzULD1Hook_12 AT %MX21256.12 : BOOL;
	bArm2HorzULD1Hook_13 AT %MX21256.13 : BOOL;
	bArm2HorzULD1Hook_14 AT %MX21256.14 : BOOL;
	bArm2HorzULD1Hook_15 AT %MX21256.15 : BOOL;
	bArm2HorzULD1Hook_16 AT %MX21256.16 : BOOL;
	bArm2HorzULD1Hook_17 AT %MX21256.17 : BOOL;
	bArm2HorzULD1Hook_18 AT %MX21256.18 : BOOL;
	bArm2HorzULD1Hook_19 AT %MX21256.19 : BOOL;
	bArm2HorzULD1Hook_20 AT %MX21256.20 : BOOL;
	bArm2HorzULD1Hook_21 AT %MX21256.21 : BOOL;
	bArm2HorzULD1Hook_22 AT %MX21256.22 : BOOL;
	bArm2HorzULD1Hook_23 AT %MX21256.23 : BOOL;
	bArm2HorzULD1Hook_24 AT %MX21256.24 : BOOL;
	bArm2HorzULD1Hook_25 AT %MX21256.25 : BOOL;
	bArm2HorzULD1Hook_26 AT %MX21256.26 : BOOL;
	bArm2HorzULD1Hook_27 AT %MX21256.27 : BOOL;
	bArm2HorzULD1Hook_28 AT %MX21256.28 : BOOL;
	bArm2HorzULD1Hook_29 AT %MX21256.29 : BOOL;
	bArm2HorzULD1Hook_30 AT %MX21256.30 : BOOL;
	bArm2HorzULD1Hook_31 AT %MX21256.31 : BOOL;

	bArm2HorzStn1Hook_00 AT %MX21204.0 : BOOL;
	bArm2HorzStn1Hook_01 AT %MX21204.1 : BOOL;
	bArm2HorzStn1Hook_02 AT %MX21204.2 : BOOL;
	bArm2HorzStn1Hook_03 AT %MX21204.3 : BOOL;
	bArm2HorzStn1Hook_04 AT %MX21204.4 : BOOL;
	bArm2HorzStn1Hook_05 AT %MX21204.5 : BOOL;
	bArm2HorzStn1Hook_06 AT %MX21204.6 : BOOL;
	bArm2HorzStn1Hook_07 AT %MX21204.7 : BOOL;
	bArm2HorzStn1Hook_08 AT %MX21204.8 : BOOL;
	bArm2HorzStn1Hook_09 AT %MX21204.9 : BOOL;
	bArm2HorzStn1Hook_10 AT %MX21204.10 : BOOL;
	bArm2HorzStn1Hook_11 AT %MX21204.11 : BOOL;
	bArm2HorzStn1Hook_12 AT %MX21204.12 : BOOL;
	bArm2HorzStn1Hook_13 AT %MX21204.13 : BOOL;
	bArm2HorzStn1Hook_14 AT %MX21204.14 : BOOL;
	bArm2HorzStn1Hook_15 AT %MX21204.15 : BOOL;
	bArm2HorzStn1Hook_16 AT %MX21204.16 : BOOL;
	bArm2HorzStn1Hook_17 AT %MX21204.17 : BOOL;
	bArm2HorzStn1Hook_18 AT %MX21204.18 : BOOL;
	bArm2HorzStn1Hook_19 AT %MX21204.19 : BOOL;
	bArm2HorzStn1Hook_20 AT %MX21204.20 : BOOL;
	bArm2HorzStn1Hook_21 AT %MX21204.21 : BOOL;
	bArm2HorzStn1Hook_22 AT %MX21204.22 : BOOL;
	bArm2HorzStn1Hook_23 AT %MX21204.23 : BOOL;
	bArm2HorzStn1Hook_24 AT %MX21204.24 : BOOL;
	bArm2HorzStn1Hook_25 AT %MX21204.25 : BOOL;
	bArm2HorzStn1Hook_26 AT %MX21204.26 : BOOL;
	bArm2HorzStn1Hook_27 AT %MX21204.27 : BOOL;
	bArm2HorzStn1Hook_28 AT %MX21204.28 : BOOL;
	bArm2HorzStn1Hook_29 AT %MX21204.29 : BOOL;
	bArm2HorzStn1Hook_30 AT %MX21204.30 : BOOL;
	bArm2HorzStn1Hook_31 AT %MX21204.31 : BOOL;

	bArm2HorzStn2Hook_00 AT %MX21208.0 : BOOL;
	bArm2HorzStn2Hook_01 AT %MX21208.1 : BOOL;
	bArm2HorzStn2Hook_02 AT %MX21208.2 : BOOL;
	bArm2HorzStn2Hook_03 AT %MX21208.3 : BOOL;
	bArm2HorzStn2Hook_04 AT %MX21208.4 : BOOL;
	bArm2HorzStn2Hook_05 AT %MX21208.5 : BOOL;
	bArm2HorzStn2Hook_06 AT %MX21208.6 : BOOL;
	bArm2HorzStn2Hook_07 AT %MX21208.7 : BOOL;
	bArm2HorzStn2Hook_08 AT %MX21208.8 : BOOL;
	bArm2HorzStn2Hook_09 AT %MX21208.9 : BOOL;
	bArm2HorzStn2Hook_10 AT %MX21208.10 : BOOL;
	bArm2HorzStn2Hook_11 AT %MX21208.11 : BOOL;
	bArm2HorzStn2Hook_12 AT %MX21208.12 : BOOL;
	bArm2HorzStn2Hook_13 AT %MX21208.13 : BOOL;
	bArm2HorzStn2Hook_14 AT %MX21208.14 : BOOL;
	bArm2HorzStn2Hook_15 AT %MX21208.15 : BOOL;
	bArm2HorzStn2Hook_16 AT %MX21208.16 : BOOL;
	bArm2HorzStn2Hook_17 AT %MX21208.17 : BOOL;
	bArm2HorzStn2Hook_18 AT %MX21208.18 : BOOL;
	bArm2HorzStn2Hook_19 AT %MX21208.19 : BOOL;
	bArm2HorzStn2Hook_20 AT %MX21208.20 : BOOL;
	bArm2HorzStn2Hook_21 AT %MX21208.21 : BOOL;
	bArm2HorzStn2Hook_22 AT %MX21208.22 : BOOL;
	bArm2HorzStn2Hook_23 AT %MX21208.23 : BOOL;
	bArm2HorzStn2Hook_24 AT %MX21208.24 : BOOL;
	bArm2HorzStn2Hook_25 AT %MX21208.25 : BOOL;
	bArm2HorzStn2Hook_26 AT %MX21208.26 : BOOL;
	bArm2HorzStn2Hook_27 AT %MX21208.27 : BOOL;
	bArm2HorzStn2Hook_28 AT %MX21208.28 : BOOL;
	bArm2HorzStn2Hook_29 AT %MX21208.29 : BOOL;
	bArm2HorzStn2Hook_30 AT %MX21208.30 : BOOL;
	bArm2HorzStn2Hook_31 AT %MX21208.31 : BOOL;

	bArm2HorzStn3Hook_00 AT %MX21212.0 : BOOL;
	bArm2HorzStn3Hook_01 AT %MX21212.1 : BOOL;
	bArm2HorzStn3Hook_02 AT %MX21212.2 : BOOL;
	bArm2HorzStn3Hook_03 AT %MX21212.3 : BOOL;
	bArm2HorzStn3Hook_04 AT %MX21212.4 : BOOL;
	bArm2HorzStn3Hook_05 AT %MX21212.5 : BOOL;
	bArm2HorzStn3Hook_06 AT %MX21212.6 : BOOL;
	bArm2HorzStn3Hook_07 AT %MX21212.7 : BOOL;
	bArm2HorzStn3Hook_08 AT %MX21212.8 : BOOL;
	bArm2HorzStn3Hook_09 AT %MX21212.9 : BOOL;
	bArm2HorzStn3Hook_10 AT %MX21212.10 : BOOL;
	bArm2HorzStn3Hook_11 AT %MX21212.11 : BOOL;
	bArm2HorzStn3Hook_12 AT %MX21212.12 : BOOL;
	bArm2HorzStn3Hook_13 AT %MX21212.13 : BOOL;
	bArm2HorzStn3Hook_14 AT %MX21212.14 : BOOL;
	bArm2HorzStn3Hook_15 AT %MX21212.15 : BOOL;
	bArm2HorzStn3Hook_16 AT %MX21212.16 : BOOL;
	bArm2HorzStn3Hook_17 AT %MX21212.17 : BOOL;
	bArm2HorzStn3Hook_18 AT %MX21212.18 : BOOL;
	bArm2HorzStn3Hook_19 AT %MX21212.19 : BOOL;
	bArm2HorzStn3Hook_20 AT %MX21212.20 : BOOL;
	bArm2HorzStn3Hook_21 AT %MX21212.21 : BOOL;
	bArm2HorzStn3Hook_22 AT %MX21212.22 : BOOL;
	bArm2HorzStn3Hook_23 AT %MX21212.23 : BOOL;
	bArm2HorzStn3Hook_24 AT %MX21212.24 : BOOL;
	bArm2HorzStn3Hook_25 AT %MX21212.25 : BOOL;
	bArm2HorzStn3Hook_26 AT %MX21212.26 : BOOL;
	bArm2HorzStn3Hook_27 AT %MX21212.27 : BOOL;
	bArm2HorzStn3Hook_28 AT %MX21212.28 : BOOL;
	bArm2HorzStn3Hook_29 AT %MX21212.29 : BOOL;
	bArm2HorzStn3Hook_30 AT %MX21212.30 : BOOL;
	bArm2HorzStn3Hook_31 AT %MX21212.31 : BOOL;

	bArm2HorzStn4Hook_00 AT %MX21216.0 : BOOL;
	bArm2HorzStn4Hook_01 AT %MX21216.1 : BOOL;
	bArm2HorzStn4Hook_02 AT %MX21216.2 : BOOL;
	bArm2HorzStn4Hook_03 AT %MX21216.3 : BOOL;
	bArm2HorzStn4Hook_04 AT %MX21216.4 : BOOL;
	bArm2HorzStn4Hook_05 AT %MX21216.5 : BOOL;
	bArm2HorzStn4Hook_06 AT %MX21216.6 : BOOL;
	bArm2HorzStn4Hook_07 AT %MX21216.7 : BOOL;
	bArm2HorzStn4Hook_08 AT %MX21216.8 : BOOL;
	bArm2HorzStn4Hook_09 AT %MX21216.9 : BOOL;
	bArm2HorzStn4Hook_10 AT %MX21216.10 : BOOL;
	bArm2HorzStn4Hook_11 AT %MX21216.11 : BOOL;
	bArm2HorzStn4Hook_12 AT %MX21216.12 : BOOL;
	bArm2HorzStn4Hook_13 AT %MX21216.13 : BOOL;
	bArm2HorzStn4Hook_14 AT %MX21216.14 : BOOL;
	bArm2HorzStn4Hook_15 AT %MX21216.15 : BOOL;
	bArm2HorzStn4Hook_16 AT %MX21216.16 : BOOL;
	bArm2HorzStn4Hook_17 AT %MX21216.17 : BOOL;
	bArm2HorzStn4Hook_18 AT %MX21216.18 : BOOL;
	bArm2HorzStn4Hook_19 AT %MX21216.19 : BOOL;
	bArm2HorzStn4Hook_20 AT %MX21216.20 : BOOL;
	bArm2HorzStn4Hook_21 AT %MX21216.21 : BOOL;
	bArm2HorzStn4Hook_22 AT %MX21216.22 : BOOL;
	bArm2HorzStn4Hook_23 AT %MX21216.23 : BOOL;
	bArm2HorzStn4Hook_24 AT %MX21216.24 : BOOL;
	bArm2HorzStn4Hook_25 AT %MX21216.25 : BOOL;
	bArm2HorzStn4Hook_26 AT %MX21216.26 : BOOL;
	bArm2HorzStn4Hook_27 AT %MX21216.27 : BOOL;
	bArm2HorzStn4Hook_28 AT %MX21216.28 : BOOL;
	bArm2HorzStn4Hook_29 AT %MX21216.29 : BOOL;
	bArm2HorzStn4Hook_30 AT %MX21216.30 : BOOL;
	bArm2HorzStn4Hook_31 AT %MX21216.31 : BOOL;

	bArm2HorzStn5Hook_00 AT %MX21220.0 : BOOL;
	bArm2HorzStn5Hook_01 AT %MX21220.1 : BOOL;
	bArm2HorzStn5Hook_02 AT %MX21220.2 : BOOL;
	bArm2HorzStn5Hook_03 AT %MX21220.3 : BOOL;
	bArm2HorzStn5Hook_04 AT %MX21220.4 : BOOL;
	bArm2HorzStn5Hook_05 AT %MX21220.5 : BOOL;
	bArm2HorzStn5Hook_06 AT %MX21220.6 : BOOL;
	bArm2HorzStn5Hook_07 AT %MX21220.7 : BOOL;
	bArm2HorzStn5Hook_08 AT %MX21220.8 : BOOL;
	bArm2HorzStn5Hook_09 AT %MX21220.9 : BOOL;
	bArm2HorzStn5Hook_10 AT %MX21220.10 : BOOL;
	bArm2HorzStn5Hook_11 AT %MX21220.11 : BOOL;
	bArm2HorzStn5Hook_12 AT %MX21220.12 : BOOL;
	bArm2HorzStn5Hook_13 AT %MX21220.13 : BOOL;
	bArm2HorzStn5Hook_14 AT %MX21220.14 : BOOL;
	bArm2HorzStn5Hook_15 AT %MX21220.15 : BOOL;
	bArm2HorzStn5Hook_16 AT %MX21220.16 : BOOL;
	bArm2HorzStn5Hook_17 AT %MX21220.17 : BOOL;
	bArm2HorzStn5Hook_18 AT %MX21220.18 : BOOL;
	bArm2HorzStn5Hook_19 AT %MX21220.19 : BOOL;
	bArm2HorzStn5Hook_20 AT %MX21220.20 : BOOL;
	bArm2HorzStn5Hook_21 AT %MX21220.21 : BOOL;
	bArm2HorzStn5Hook_22 AT %MX21220.22 : BOOL;
	bArm2HorzStn5Hook_23 AT %MX21220.23 : BOOL;
	bArm2HorzStn5Hook_24 AT %MX21220.24 : BOOL;
	bArm2HorzStn5Hook_25 AT %MX21220.25 : BOOL;
	bArm2HorzStn5Hook_26 AT %MX21220.26 : BOOL;
	bArm2HorzStn5Hook_27 AT %MX21220.27 : BOOL;
	bArm2HorzStn5Hook_28 AT %MX21220.28 : BOOL;
	bArm2HorzStn5Hook_29 AT %MX21220.29 : BOOL;
	bArm2HorzStn5Hook_30 AT %MX21220.30 : BOOL;
	bArm2HorzStn5Hook_31 AT %MX21220.31 : BOOL;

	bArm2HorzStn6Hook_00 AT %MX21224.0 : BOOL;
	bArm2HorzStn6Hook_01 AT %MX21224.1 : BOOL;
	bArm2HorzStn6Hook_02 AT %MX21224.2 : BOOL;
	bArm2HorzStn6Hook_03 AT %MX21224.3 : BOOL;
	bArm2HorzStn6Hook_04 AT %MX21224.4 : BOOL;
	bArm2HorzStn6Hook_05 AT %MX21224.5 : BOOL;
	bArm2HorzStn6Hook_06 AT %MX21224.6 : BOOL;
	bArm2HorzStn6Hook_07 AT %MX21224.7 : BOOL;
	bArm2HorzStn6Hook_08 AT %MX21224.8 : BOOL;
	bArm2HorzStn6Hook_09 AT %MX21224.9 : BOOL;
	bArm2HorzStn6Hook_10 AT %MX21224.10 : BOOL;
	bArm2HorzStn6Hook_11 AT %MX21224.11 : BOOL;
	bArm2HorzStn6Hook_12 AT %MX21224.12 : BOOL;
	bArm2HorzStn6Hook_13 AT %MX21224.13 : BOOL;
	bArm2HorzStn6Hook_14 AT %MX21224.14 : BOOL;
	bArm2HorzStn6Hook_15 AT %MX21224.15 : BOOL;
	bArm2HorzStn6Hook_16 AT %MX21224.16 : BOOL;
	bArm2HorzStn6Hook_17 AT %MX21224.17 : BOOL;
	bArm2HorzStn6Hook_18 AT %MX21224.18 : BOOL;
	bArm2HorzStn6Hook_19 AT %MX21224.19 : BOOL;
	bArm2HorzStn6Hook_20 AT %MX21224.20 : BOOL;
	bArm2HorzStn6Hook_21 AT %MX21224.21 : BOOL;
	bArm2HorzStn6Hook_22 AT %MX21224.22 : BOOL;
	bArm2HorzStn6Hook_23 AT %MX21224.23 : BOOL;
	bArm2HorzStn6Hook_24 AT %MX21224.24 : BOOL;
	bArm2HorzStn6Hook_25 AT %MX21224.25 : BOOL;
	bArm2HorzStn6Hook_26 AT %MX21224.26 : BOOL;
	bArm2HorzStn6Hook_27 AT %MX21224.27 : BOOL;
	bArm2HorzStn6Hook_28 AT %MX21224.28 : BOOL;
	bArm2HorzStn6Hook_29 AT %MX21224.29 : BOOL;
	bArm2HorzStn6Hook_30 AT %MX21224.30 : BOOL;
	bArm2HorzStn6Hook_31 AT %MX21224.31 : BOOL;

	bArm2HorzStn7Hook_00 AT %MX21228.0 : BOOL;
	bArm2HorzStn7Hook_01 AT %MX21228.1 : BOOL;
	bArm2HorzStn7Hook_02 AT %MX21228.2 : BOOL;
	bArm2HorzStn7Hook_03 AT %MX21228.3 : BOOL;
	bArm2HorzStn7Hook_04 AT %MX21228.4 : BOOL;
	bArm2HorzStn7Hook_05 AT %MX21228.5 : BOOL;
	bArm2HorzStn7Hook_06 AT %MX21228.6 : BOOL;
	bArm2HorzStn7Hook_07 AT %MX21228.7 : BOOL;
	bArm2HorzStn7Hook_08 AT %MX21228.8 : BOOL;
	bArm2HorzStn7Hook_09 AT %MX21228.9 : BOOL;
	bArm2HorzStn7Hook_10 AT %MX21228.10 : BOOL;
	bArm2HorzStn7Hook_11 AT %MX21228.11 : BOOL;
	bArm2HorzStn7Hook_12 AT %MX21228.12 : BOOL;
	bArm2HorzStn7Hook_13 AT %MX21228.13 : BOOL;
	bArm2HorzStn7Hook_14 AT %MX21228.14 : BOOL;
	bArm2HorzStn7Hook_15 AT %MX21228.15 : BOOL;
	bArm2HorzStn7Hook_16 AT %MX21228.16 : BOOL;
	bArm2HorzStn7Hook_17 AT %MX21228.17 : BOOL;
	bArm2HorzStn7Hook_18 AT %MX21228.18 : BOOL;
	bArm2HorzStn7Hook_19 AT %MX21228.19 : BOOL;
	bArm2HorzStn7Hook_20 AT %MX21228.20 : BOOL;
	bArm2HorzStn7Hook_21 AT %MX21228.21 : BOOL;
	bArm2HorzStn7Hook_22 AT %MX21228.22 : BOOL;
	bArm2HorzStn7Hook_23 AT %MX21228.23 : BOOL;
	bArm2HorzStn7Hook_24 AT %MX21228.24 : BOOL;
	bArm2HorzStn7Hook_25 AT %MX21228.25 : BOOL;
	bArm2HorzStn7Hook_26 AT %MX21228.26 : BOOL;
	bArm2HorzStn7Hook_27 AT %MX21228.27 : BOOL;
	bArm2HorzStn7Hook_28 AT %MX21228.28 : BOOL;
	bArm2HorzStn7Hook_29 AT %MX21228.29 : BOOL;
	bArm2HorzStn7Hook_30 AT %MX21228.30 : BOOL;
	bArm2HorzStn7Hook_31 AT %MX21228.31 : BOOL;

	bArm2HorzStn8Hook_00 AT %MX21232.0 : BOOL;
	bArm2HorzStn8Hook_01 AT %MX21232.1 : BOOL;
	bArm2HorzStn8Hook_02 AT %MX21232.2 : BOOL;
	bArm2HorzStn8Hook_03 AT %MX21232.3 : BOOL;
	bArm2HorzStn8Hook_04 AT %MX21232.4 : BOOL;
	bArm2HorzStn8Hook_05 AT %MX21232.5 : BOOL;
	bArm2HorzStn8Hook_06 AT %MX21232.6 : BOOL;
	bArm2HorzStn8Hook_07 AT %MX21232.7 : BOOL;
	bArm2HorzStn8Hook_08 AT %MX21232.8 : BOOL;
	bArm2HorzStn8Hook_09 AT %MX21232.9 : BOOL;
	bArm2HorzStn8Hook_10 AT %MX21232.10 : BOOL;
	bArm2HorzStn8Hook_11 AT %MX21232.11 : BOOL;
	bArm2HorzStn8Hook_12 AT %MX21232.12 : BOOL;
	bArm2HorzStn8Hook_13 AT %MX21232.13 : BOOL;
	bArm2HorzStn8Hook_14 AT %MX21232.14 : BOOL;
	bArm2HorzStn8Hook_15 AT %MX21232.15 : BOOL;
	bArm2HorzStn8Hook_16 AT %MX21232.16 : BOOL;
	bArm2HorzStn8Hook_17 AT %MX21232.17 : BOOL;
	bArm2HorzStn8Hook_18 AT %MX21232.18 : BOOL;
	bArm2HorzStn8Hook_19 AT %MX21232.19 : BOOL;
	bArm2HorzStn8Hook_20 AT %MX21232.20 : BOOL;
	bArm2HorzStn8Hook_21 AT %MX21232.21 : BOOL;
	bArm2HorzStn8Hook_22 AT %MX21232.22 : BOOL;
	bArm2HorzStn8Hook_23 AT %MX21232.23 : BOOL;
	bArm2HorzStn8Hook_24 AT %MX21232.24 : BOOL;
	bArm2HorzStn8Hook_25 AT %MX21232.25 : BOOL;
	bArm2HorzStn8Hook_26 AT %MX21232.26 : BOOL;
	bArm2HorzStn8Hook_27 AT %MX21232.27 : BOOL;
	bArm2HorzStn8Hook_28 AT %MX21232.28 : BOOL;
	bArm2HorzStn8Hook_29 AT %MX21232.29 : BOOL;
	bArm2HorzStn8Hook_30 AT %MX21232.30 : BOOL;
	bArm2HorzStn8Hook_31 AT %MX21232.31 : BOOL;

	bArm2HorzStn9Hook_00 AT %MX21236.0 : BOOL;
	bArm2HorzStn9Hook_01 AT %MX21236.1 : BOOL;
	bArm2HorzStn9Hook_02 AT %MX21236.2 : BOOL;
	bArm2HorzStn9Hook_03 AT %MX21236.3 : BOOL;
	bArm2HorzStn9Hook_04 AT %MX21236.4 : BOOL;
	bArm2HorzStn9Hook_05 AT %MX21236.5 : BOOL;
	bArm2HorzStn9Hook_06 AT %MX21236.6 : BOOL;
	bArm2HorzStn9Hook_07 AT %MX21236.7 : BOOL;
	bArm2HorzStn9Hook_08 AT %MX21236.8 : BOOL;
	bArm2HorzStn9Hook_09 AT %MX21236.9 : BOOL;
	bArm2HorzStn9Hook_10 AT %MX21236.10 : BOOL;
	bArm2HorzStn9Hook_11 AT %MX21236.11 : BOOL;
	bArm2HorzStn9Hook_12 AT %MX21236.12 : BOOL;
	bArm2HorzStn9Hook_13 AT %MX21236.13 : BOOL;
	bArm2HorzStn9Hook_14 AT %MX21236.14 : BOOL;
	bArm2HorzStn9Hook_15 AT %MX21236.15 : BOOL;
	bArm2HorzStn9Hook_16 AT %MX21236.16 : BOOL;
	bArm2HorzStn9Hook_17 AT %MX21236.17 : BOOL;
	bArm2HorzStn9Hook_18 AT %MX21236.18 : BOOL;
	bArm2HorzStn9Hook_19 AT %MX21236.19 : BOOL;
	bArm2HorzStn9Hook_20 AT %MX21236.20 : BOOL;
	bArm2HorzStn9Hook_21 AT %MX21236.21 : BOOL;
	bArm2HorzStn9Hook_22 AT %MX21236.22 : BOOL;
	bArm2HorzStn9Hook_23 AT %MX21236.23 : BOOL;
	bArm2HorzStn9Hook_24 AT %MX21236.24 : BOOL;
	bArm2HorzStn9Hook_25 AT %MX21236.25 : BOOL;
	bArm2HorzStn9Hook_26 AT %MX21236.26 : BOOL;
	bArm2HorzStn9Hook_27 AT %MX21236.27 : BOOL;
	bArm2HorzStn9Hook_28 AT %MX21236.28 : BOOL;
	bArm2HorzStn9Hook_29 AT %MX21236.29 : BOOL;
	bArm2HorzStn9Hook_30 AT %MX21236.30 : BOOL;
	bArm2HorzStn9Hook_31 AT %MX21236.31 : BOOL;

	bArm2HorzStn10Hook_00 AT %MX21240.0 : BOOL;
	bArm2HorzStn10Hook_01 AT %MX21240.1 : BOOL;
	bArm2HorzStn10Hook_02 AT %MX21240.2 : BOOL;
	bArm2HorzStn10Hook_03 AT %MX21240.3 : BOOL;
	bArm2HorzStn10Hook_04 AT %MX21240.4 : BOOL;
	bArm2HorzStn10Hook_05 AT %MX21240.5 : BOOL;
	bArm2HorzStn10Hook_06 AT %MX21240.6 : BOOL;
	bArm2HorzStn10Hook_07 AT %MX21240.7 : BOOL;
	bArm2HorzStn10Hook_08 AT %MX21240.8 : BOOL;
	bArm2HorzStn10Hook_09 AT %MX21240.9 : BOOL;
	bArm2HorzStn10Hook_10 AT %MX21240.10 : BOOL;
	bArm2HorzStn10Hook_11 AT %MX21240.11 : BOOL;
	bArm2HorzStn10Hook_12 AT %MX21240.12 : BOOL;
	bArm2HorzStn10Hook_13 AT %MX21240.13 : BOOL;
	bArm2HorzStn10Hook_14 AT %MX21240.14 : BOOL;
	bArm2HorzStn10Hook_15 AT %MX21240.15 : BOOL;
	bArm2HorzStn10Hook_16 AT %MX21240.16 : BOOL;
	bArm2HorzStn10Hook_17 AT %MX21240.17 : BOOL;
	bArm2HorzStn10Hook_18 AT %MX21240.18 : BOOL;
	bArm2HorzStn10Hook_19 AT %MX21240.19 : BOOL;
	bArm2HorzStn10Hook_20 AT %MX21240.20 : BOOL;
	bArm2HorzStn10Hook_21 AT %MX21240.21 : BOOL;
	bArm2HorzStn10Hook_22 AT %MX21240.22 : BOOL;
	bArm2HorzStn10Hook_23 AT %MX21240.23 : BOOL;
	bArm2HorzStn10Hook_24 AT %MX21240.24 : BOOL;
	bArm2HorzStn10Hook_25 AT %MX21240.25 : BOOL;
	bArm2HorzStn10Hook_26 AT %MX21240.26 : BOOL;
	bArm2HorzStn10Hook_27 AT %MX21240.27 : BOOL;
	bArm2HorzStn10Hook_28 AT %MX21240.28 : BOOL;
	bArm2HorzStn10Hook_29 AT %MX21240.29 : BOOL;
	bArm2HorzStn10Hook_30 AT %MX21240.30 : BOOL;
	bArm2HorzStn10Hook_31 AT %MX21240.31 : BOOL;

	bArm2HorzStn11Hook_00 AT %MX21244.0 : BOOL;
	bArm2HorzStn11Hook_01 AT %MX21244.1 : BOOL;
	bArm2HorzStn11Hook_02 AT %MX21244.2 : BOOL;
	bArm2HorzStn11Hook_03 AT %MX21244.3 : BOOL;
	bArm2HorzStn11Hook_04 AT %MX21244.4 : BOOL;
	bArm2HorzStn11Hook_05 AT %MX21244.5 : BOOL;
	bArm2HorzStn11Hook_06 AT %MX21244.6 : BOOL;
	bArm2HorzStn11Hook_07 AT %MX21244.7 : BOOL;
	bArm2HorzStn11Hook_08 AT %MX21244.8 : BOOL;
	bArm2HorzStn11Hook_09 AT %MX21244.9 : BOOL;
	bArm2HorzStn11Hook_10 AT %MX21244.10 : BOOL;
	bArm2HorzStn11Hook_11 AT %MX21244.11 : BOOL;
	bArm2HorzStn11Hook_12 AT %MX21244.12 : BOOL;
	bArm2HorzStn11Hook_13 AT %MX21244.13 : BOOL;
	bArm2HorzStn11Hook_14 AT %MX21244.14 : BOOL;
	bArm2HorzStn11Hook_15 AT %MX21244.15 : BOOL;
	bArm2HorzStn11Hook_16 AT %MX21244.16 : BOOL;
	bArm2HorzStn11Hook_17 AT %MX21244.17 : BOOL;
	bArm2HorzStn11Hook_18 AT %MX21244.18 : BOOL;
	bArm2HorzStn11Hook_19 AT %MX21244.19 : BOOL;
	bArm2HorzStn11Hook_20 AT %MX21244.20 : BOOL;
	bArm2HorzStn11Hook_21 AT %MX21244.21 : BOOL;
	bArm2HorzStn11Hook_22 AT %MX21244.22 : BOOL;
	bArm2HorzStn11Hook_23 AT %MX21244.23 : BOOL;
	bArm2HorzStn11Hook_24 AT %MX21244.24 : BOOL;
	bArm2HorzStn11Hook_25 AT %MX21244.25 : BOOL;
	bArm2HorzStn11Hook_26 AT %MX21244.26 : BOOL;
	bArm2HorzStn11Hook_27 AT %MX21244.27 : BOOL;
	bArm2HorzStn11Hook_28 AT %MX21244.28 : BOOL;
	bArm2HorzStn11Hook_29 AT %MX21244.29 : BOOL;
	bArm2HorzStn11Hook_30 AT %MX21244.30 : BOOL;
	bArm2HorzStn11Hook_31 AT %MX21244.31 : BOOL;

	bArm2HorzStn12Hook_00 AT %MX21248.0 : BOOL;
	bArm2HorzStn12Hook_01 AT %MX21248.1 : BOOL;
	bArm2HorzStn12Hook_02 AT %MX21248.2 : BOOL;
	bArm2HorzStn12Hook_03 AT %MX21248.3 : BOOL;
	bArm2HorzStn12Hook_04 AT %MX21248.4 : BOOL;
	bArm2HorzStn12Hook_05 AT %MX21248.5 : BOOL;
	bArm2HorzStn12Hook_06 AT %MX21248.6 : BOOL;
	bArm2HorzStn12Hook_07 AT %MX21248.7 : BOOL;
	bArm2HorzStn12Hook_08 AT %MX21248.8 : BOOL;
	bArm2HorzStn12Hook_09 AT %MX21248.9 : BOOL;
	bArm2HorzStn12Hook_10 AT %MX21248.10 : BOOL;
	bArm2HorzStn12Hook_11 AT %MX21248.11 : BOOL;
	bArm2HorzStn12Hook_12 AT %MX21248.12 : BOOL;
	bArm2HorzStn12Hook_13 AT %MX21248.13 : BOOL;
	bArm2HorzStn12Hook_14 AT %MX21248.14 : BOOL;
	bArm2HorzStn12Hook_15 AT %MX21248.15 : BOOL;
	bArm2HorzStn12Hook_16 AT %MX21248.16 : BOOL;
	bArm2HorzStn12Hook_17 AT %MX21248.17 : BOOL;
	bArm2HorzStn12Hook_18 AT %MX21248.18 : BOOL;
	bArm2HorzStn12Hook_19 AT %MX21248.19 : BOOL;
	bArm2HorzStn12Hook_20 AT %MX21248.20 : BOOL;
	bArm2HorzStn12Hook_21 AT %MX21248.21 : BOOL;
	bArm2HorzStn12Hook_22 AT %MX21248.22 : BOOL;
	bArm2HorzStn12Hook_23 AT %MX21248.23 : BOOL;
	bArm2HorzStn12Hook_24 AT %MX21248.24 : BOOL;
	bArm2HorzStn12Hook_25 AT %MX21248.25 : BOOL;
	bArm2HorzStn12Hook_26 AT %MX21248.26 : BOOL;
	bArm2HorzStn12Hook_27 AT %MX21248.27 : BOOL;
	bArm2HorzStn12Hook_28 AT %MX21248.28 : BOOL;
	bArm2HorzStn12Hook_29 AT %MX21248.29 : BOOL;
	bArm2HorzStn12Hook_30 AT %MX21248.30 : BOOL;
	bArm2HorzStn12Hook_31 AT %MX21248.31 : BOOL;

(* xxxxxxxxxxxxxxxxxxxxxxxxxxxxxxxxxxxxxxx Unhook word xxxxxxxxxxxxxxxxxxxxxxxxxxxxxxxxxxxxxxx*)
(*====================== Unhook BOOL LINK with %MX21300-MX21399 ======================*)

	bArm2HorzLD1Unhook_00 AT %MX21352.0 : BOOL;
	bArm2HorzLD1Unhook_01 AT %MX21352.1 : BOOL;
	bArm2HorzLD1Unhook_02 AT %MX21352.2 : BOOL;
	bArm2HorzLD1Unhook_03 AT %MX21352.3 : BOOL;
	bArm2HorzLD1Unhook_04 AT %MX21352.4 : BOOL;
	bArm2HorzLD1Unhook_05 AT %MX21352.5 : BOOL;
	bArm2HorzLD1Unhook_06 AT %MX21352.6 : BOOL;
	bArm2HorzLD1Unhook_07 AT %MX21352.7 : BOOL;
	bArm2HorzLD1Unhook_08 AT %MX21352.8 : BOOL;
	bArm2HorzLD1Unhook_09 AT %MX21352.9 : BOOL;
	bArm2HorzLD1Unhook_10 AT %MX21352.10 : BOOL;
	bArm2HorzLD1Unhook_11 AT %MX21352.11 : BOOL;
	bArm2HorzLD1Unhook_12 AT %MX21352.12 : BOOL;
	bArm2HorzLD1Unhook_13 AT %MX21352.13 : BOOL;
	bArm2HorzLD1Unhook_14 AT %MX21352.14 : BOOL;
	bArm2HorzLD1Unhook_15 AT %MX21352.15 : BOOL;
	bArm2HorzLD1Unhook_16 AT %MX21352.16 : BOOL;
	bArm2HorzLD1Unhook_17 AT %MX21352.17 : BOOL;
	bArm2HorzLD1Unhook_18 AT %MX21352.18 : BOOL;
	bArm2HorzLD1Unhook_19 AT %MX21352.19 : BOOL;
	bArm2HorzLD1Unhook_20 AT %MX21352.20 : BOOL;
	bArm2HorzLD1Unhook_21 AT %MX21352.21 : BOOL;
	bArm2HorzLD1Unhook_22 AT %MX21352.22 : BOOL;
	bArm2HorzLD1Unhook_23 AT %MX21352.23 : BOOL;
	bArm2HorzLD1Unhook_24 AT %MX21352.24 : BOOL;
	bArm2HorzLD1Unhook_25 AT %MX21352.25 : BOOL;
	bArm2HorzLD1Unhook_26 AT %MX21352.26 : BOOL;
	bArm2HorzLD1Unhook_27 AT %MX21352.27 : BOOL;
	bArm2HorzLD1Unhook_28 AT %MX21352.28 : BOOL;
	bArm2HorzLD1Unhook_29 AT %MX21352.29 : BOOL;
	bArm2HorzLD1Unhook_30 AT %MX21352.30 : BOOL;
	bArm2HorzLD1Unhook_31 AT %MX21352.31 : BOOL;

	bArm2HorzULD1Unhook_00 AT %MX21356.0 : BOOL;
	bArm2HorzULD1Unhook_01 AT %MX21356.1 : BOOL;
	bArm2HorzULD1Unhook_02 AT %MX21356.2 : BOOL;
	bArm2HorzULD1Unhook_03 AT %MX21356.3 : BOOL;
	bArm2HorzULD1Unhook_04 AT %MX21356.4 : BOOL;
	bArm2HorzULD1Unhook_05 AT %MX21356.5 : BOOL;
	bArm2HorzULD1Unhook_06 AT %MX21356.6 : BOOL;
	bArm2HorzULD1Unhook_07 AT %MX21356.7 : BOOL;
	bArm2HorzULD1Unhook_08 AT %MX21356.8 : BOOL;
	bArm2HorzULD1Unhook_09 AT %MX21356.9 : BOOL;
	bArm2HorzULD1Unhook_10 AT %MX21356.10 : BOOL;
	bArm2HorzULD1Unhook_11 AT %MX21356.11 : BOOL;
	bArm2HorzULD1Unhook_12 AT %MX21356.12 : BOOL;
	bArm2HorzULD1Unhook_13 AT %MX21356.13 : BOOL;
	bArm2HorzULD1Unhook_14 AT %MX21356.14 : BOOL;
	bArm2HorzULD1Unhook_15 AT %MX21356.15 : BOOL;
	bArm2HorzULD1Unhook_16 AT %MX21356.16 : BOOL;
	bArm2HorzULD1Unhook_17 AT %MX21356.17 : BOOL;
	bArm2HorzULD1Unhook_18 AT %MX21356.18 : BOOL;
	bArm2HorzULD1Unhook_19 AT %MX21356.19 : BOOL;
	bArm2HorzULD1Unhook_20 AT %MX21356.20 : BOOL;
	bArm2HorzULD1Unhook_21 AT %MX21356.21 : BOOL;
	bArm2HorzULD1Unhook_22 AT %MX21356.22 : BOOL;
	bArm2HorzULD1Unhook_23 AT %MX21356.23 : BOOL;
	bArm2HorzULD1Unhook_24 AT %MX21356.24 : BOOL;
	bArm2HorzULD1Unhook_25 AT %MX21356.25 : BOOL;
	bArm2HorzULD1Unhook_26 AT %MX21356.26 : BOOL;
	bArm2HorzULD1Unhook_27 AT %MX21356.27 : BOOL;
	bArm2HorzULD1Unhook_28 AT %MX21356.28 : BOOL;
	bArm2HorzULD1Unhook_29 AT %MX21356.29 : BOOL;
	bArm2HorzULD1Unhook_30 AT %MX21356.30 : BOOL;
	bArm2HorzULD1Unhook_31 AT %MX21356.31 : BOOL;

	bArm2HorzStn1Unhook_00 AT %MX21304.0 : BOOL;
	bArm2HorzStn1Unhook_01 AT %MX21304.1 : BOOL;
	bArm2HorzStn1Unhook_02 AT %MX21304.2 : BOOL;
	bArm2HorzStn1Unhook_03 AT %MX21304.3 : BOOL;
	bArm2HorzStn1Unhook_04 AT %MX21304.4 : BOOL;
	bArm2HorzStn1Unhook_05 AT %MX21304.5 : BOOL;
	bArm2HorzStn1Unhook_06 AT %MX21304.6 : BOOL;
	bArm2HorzStn1Unhook_07 AT %MX21304.7 : BOOL;
	bArm2HorzStn1Unhook_08 AT %MX21304.8 : BOOL;
	bArm2HorzStn1Unhook_09 AT %MX21304.9 : BOOL;
	bArm2HorzStn1Unhook_10 AT %MX21304.10 : BOOL;
	bArm2HorzStn1Unhook_11 AT %MX21304.11 : BOOL;
	bArm2HorzStn1Unhook_12 AT %MX21304.12 : BOOL;
	bArm2HorzStn1Unhook_13 AT %MX21304.13 : BOOL;
	bArm2HorzStn1Unhook_14 AT %MX21304.14 : BOOL;
	bArm2HorzStn1Unhook_15 AT %MX21304.15 : BOOL;
	bArm2HorzStn1Unhook_16 AT %MX21304.16 : BOOL;
	bArm2HorzStn1Unhook_17 AT %MX21304.17 : BOOL;
	bArm2HorzStn1Unhook_18 AT %MX21304.18 : BOOL;
	bArm2HorzStn1Unhook_19 AT %MX21304.19 : BOOL;
	bArm2HorzStn1Unhook_20 AT %MX21304.20 : BOOL;
	bArm2HorzStn1Unhook_21 AT %MX21304.21 : BOOL;
	bArm2HorzStn1Unhook_22 AT %MX21304.22 : BOOL;
	bArm2HorzStn1Unhook_23 AT %MX21304.23 : BOOL;
	bArm2HorzStn1Unhook_24 AT %MX21304.24 : BOOL;
	bArm2HorzStn1Unhook_25 AT %MX21304.25 : BOOL;
	bArm2HorzStn1Unhook_26 AT %MX21304.26 : BOOL;
	bArm2HorzStn1Unhook_27 AT %MX21304.27 : BOOL;
	bArm2HorzStn1Unhook_28 AT %MX21304.28 : BOOL;
	bArm2HorzStn1Unhook_29 AT %MX21304.29 : BOOL;
	bArm2HorzStn1Unhook_30 AT %MX21304.30 : BOOL;
	bArm2HorzStn1Unhook_31 AT %MX21304.31 : BOOL;

	bArm2HorzStn2Unhook_00 AT %MX21308.0 : BOOL;
	bArm2HorzStn2Unhook_01 AT %MX21308.1 : BOOL;
	bArm2HorzStn2Unhook_02 AT %MX21308.2 : BOOL;
	bArm2HorzStn2Unhook_03 AT %MX21308.3 : BOOL;
	bArm2HorzStn2Unhook_04 AT %MX21308.4 : BOOL;
	bArm2HorzStn2Unhook_05 AT %MX21308.5 : BOOL;
	bArm2HorzStn2Unhook_06 AT %MX21308.6 : BOOL;
	bArm2HorzStn2Unhook_07 AT %MX21308.7 : BOOL;
	bArm2HorzStn2Unhook_08 AT %MX21308.8 : BOOL;
	bArm2HorzStn2Unhook_09 AT %MX21308.9 : BOOL;
	bArm2HorzStn2Unhook_10 AT %MX21308.10 : BOOL;
	bArm2HorzStn2Unhook_11 AT %MX21308.11 : BOOL;
	bArm2HorzStn2Unhook_12 AT %MX21308.12 : BOOL;
	bArm2HorzStn2Unhook_13 AT %MX21308.13 : BOOL;
	bArm2HorzStn2Unhook_14 AT %MX21308.14 : BOOL;
	bArm2HorzStn2Unhook_15 AT %MX21308.15 : BOOL;
	bArm2HorzStn2Unhook_16 AT %MX21308.16 : BOOL;
	bArm2HorzStn2Unhook_17 AT %MX21308.17 : BOOL;
	bArm2HorzStn2Unhook_18 AT %MX21308.18 : BOOL;
	bArm2HorzStn2Unhook_19 AT %MX21308.19 : BOOL;
	bArm2HorzStn2Unhook_20 AT %MX21308.20 : BOOL;
	bArm2HorzStn2Unhook_21 AT %MX21308.21 : BOOL;
	bArm2HorzStn2Unhook_22 AT %MX21308.22 : BOOL;
	bArm2HorzStn2Unhook_23 AT %MX21308.23 : BOOL;
	bArm2HorzStn2Unhook_24 AT %MX21308.24 : BOOL;
	bArm2HorzStn2Unhook_25 AT %MX21308.25 : BOOL;
	bArm2HorzStn2Unhook_26 AT %MX21308.26 : BOOL;
	bArm2HorzStn2Unhook_27 AT %MX21308.27 : BOOL;
	bArm2HorzStn2Unhook_28 AT %MX21308.28 : BOOL;
	bArm2HorzStn2Unhook_29 AT %MX21308.29 : BOOL;
	bArm2HorzStn2Unhook_30 AT %MX21308.30 : BOOL;
	bArm2HorzStn2Unhook_31 AT %MX21308.31 : BOOL;

	bArm2HorzStn3Unhook_00 AT %MX21312.0 : BOOL;
	bArm2HorzStn3Unhook_01 AT %MX21312.1 : BOOL;
	bArm2HorzStn3Unhook_02 AT %MX21312.2 : BOOL;
	bArm2HorzStn3Unhook_03 AT %MX21312.3 : BOOL;
	bArm2HorzStn3Unhook_04 AT %MX21312.4 : BOOL;
	bArm2HorzStn3Unhook_05 AT %MX21312.5 : BOOL;
	bArm2HorzStn3Unhook_06 AT %MX21312.6 : BOOL;
	bArm2HorzStn3Unhook_07 AT %MX21312.7 : BOOL;
	bArm2HorzStn3Unhook_08 AT %MX21312.8 : BOOL;
	bArm2HorzStn3Unhook_09 AT %MX21312.9 : BOOL;
	bArm2HorzStn3Unhook_10 AT %MX21312.10 : BOOL;
	bArm2HorzStn3Unhook_11 AT %MX21312.11 : BOOL;
	bArm2HorzStn3Unhook_12 AT %MX21312.12 : BOOL;
	bArm2HorzStn3Unhook_13 AT %MX21312.13 : BOOL;
	bArm2HorzStn3Unhook_14 AT %MX21312.14 : BOOL;
	bArm2HorzStn3Unhook_15 AT %MX21312.15 : BOOL;
	bArm2HorzStn3Unhook_16 AT %MX21312.16 : BOOL;
	bArm2HorzStn3Unhook_17 AT %MX21312.17 : BOOL;
	bArm2HorzStn3Unhook_18 AT %MX21312.18 : BOOL;
	bArm2HorzStn3Unhook_19 AT %MX21312.19 : BOOL;
	bArm2HorzStn3Unhook_20 AT %MX21312.20 : BOOL;
	bArm2HorzStn3Unhook_21 AT %MX21312.21 : BOOL;
	bArm2HorzStn3Unhook_22 AT %MX21312.22 : BOOL;
	bArm2HorzStn3Unhook_23 AT %MX21312.23 : BOOL;
	bArm2HorzStn3Unhook_24 AT %MX21312.24 : BOOL;
	bArm2HorzStn3Unhook_25 AT %MX21312.25 : BOOL;
	bArm2HorzStn3Unhook_26 AT %MX21312.26 : BOOL;
	bArm2HorzStn3Unhook_27 AT %MX21312.27 : BOOL;
	bArm2HorzStn3Unhook_28 AT %MX21312.28 : BOOL;
	bArm2HorzStn3Unhook_29 AT %MX21312.29 : BOOL;
	bArm2HorzStn3Unhook_30 AT %MX21312.30 : BOOL;
	bArm2HorzStn3Unhook_31 AT %MX21312.31 : BOOL;

	bArm2HorzStn4Unhook_00 AT %MX21316.0 : BOOL;
	bArm2HorzStn4Unhook_01 AT %MX21316.1 : BOOL;
	bArm2HorzStn4Unhook_02 AT %MX21316.2 : BOOL;
	bArm2HorzStn4Unhook_03 AT %MX21316.3 : BOOL;
	bArm2HorzStn4Unhook_04 AT %MX21316.4 : BOOL;
	bArm2HorzStn4Unhook_05 AT %MX21316.5 : BOOL;
	bArm2HorzStn4Unhook_06 AT %MX21316.6 : BOOL;
	bArm2HorzStn4Unhook_07 AT %MX21316.7 : BOOL;
	bArm2HorzStn4Unhook_08 AT %MX21316.8 : BOOL;
	bArm2HorzStn4Unhook_09 AT %MX21316.9 : BOOL;
	bArm2HorzStn4Unhook_10 AT %MX21316.10 : BOOL;
	bArm2HorzStn4Unhook_11 AT %MX21316.11 : BOOL;
	bArm2HorzStn4Unhook_12 AT %MX21316.12 : BOOL;
	bArm2HorzStn4Unhook_13 AT %MX21316.13 : BOOL;
	bArm2HorzStn4Unhook_14 AT %MX21316.14 : BOOL;
	bArm2HorzStn4Unhook_15 AT %MX21316.15 : BOOL;
	bArm2HorzStn4Unhook_16 AT %MX21316.16 : BOOL;
	bArm2HorzStn4Unhook_17 AT %MX21316.17 : BOOL;
	bArm2HorzStn4Unhook_18 AT %MX21316.18 : BOOL;
	bArm2HorzStn4Unhook_19 AT %MX21316.19 : BOOL;
	bArm2HorzStn4Unhook_20 AT %MX21316.20 : BOOL;
	bArm2HorzStn4Unhook_21 AT %MX21316.21 : BOOL;
	bArm2HorzStn4Unhook_22 AT %MX21316.22 : BOOL;
	bArm2HorzStn4Unhook_23 AT %MX21316.23 : BOOL;
	bArm2HorzStn4Unhook_24 AT %MX21316.24 : BOOL;
	bArm2HorzStn4Unhook_25 AT %MX21316.25 : BOOL;
	bArm2HorzStn4Unhook_26 AT %MX21316.26 : BOOL;
	bArm2HorzStn4Unhook_27 AT %MX21316.27 : BOOL;
	bArm2HorzStn4Unhook_28 AT %MX21316.28 : BOOL;
	bArm2HorzStn4Unhook_29 AT %MX21316.29 : BOOL;
	bArm2HorzStn4Unhook_30 AT %MX21316.30 : BOOL;
	bArm2HorzStn4Unhook_31 AT %MX21316.31 : BOOL;

	bArm2HorzStn5Unhook_00 AT %MX21320.0 : BOOL;
	bArm2HorzStn5Unhook_01 AT %MX21320.1 : BOOL;
	bArm2HorzStn5Unhook_02 AT %MX21320.2 : BOOL;
	bArm2HorzStn5Unhook_03 AT %MX21320.3 : BOOL;
	bArm2HorzStn5Unhook_04 AT %MX21320.4 : BOOL;
	bArm2HorzStn5Unhook_05 AT %MX21320.5 : BOOL;
	bArm2HorzStn5Unhook_06 AT %MX21320.6 : BOOL;
	bArm2HorzStn5Unhook_07 AT %MX21320.7 : BOOL;
	bArm2HorzStn5Unhook_08 AT %MX21320.8 : BOOL;
	bArm2HorzStn5Unhook_09 AT %MX21320.9 : BOOL;
	bArm2HorzStn5Unhook_10 AT %MX21320.10 : BOOL;
	bArm2HorzStn5Unhook_11 AT %MX21320.11 : BOOL;
	bArm2HorzStn5Unhook_12 AT %MX21320.12 : BOOL;
	bArm2HorzStn5Unhook_13 AT %MX21320.13 : BOOL;
	bArm2HorzStn5Unhook_14 AT %MX21320.14 : BOOL;
	bArm2HorzStn5Unhook_15 AT %MX21320.15 : BOOL;
	bArm2HorzStn5Unhook_16 AT %MX21320.16 : BOOL;
	bArm2HorzStn5Unhook_17 AT %MX21320.17 : BOOL;
	bArm2HorzStn5Unhook_18 AT %MX21320.18 : BOOL;
	bArm2HorzStn5Unhook_19 AT %MX21320.19 : BOOL;
	bArm2HorzStn5Unhook_20 AT %MX21320.20 : BOOL;
	bArm2HorzStn5Unhook_21 AT %MX21320.21 : BOOL;
	bArm2HorzStn5Unhook_22 AT %MX21320.22 : BOOL;
	bArm2HorzStn5Unhook_23 AT %MX21320.23 : BOOL;
	bArm2HorzStn5Unhook_24 AT %MX21320.24 : BOOL;
	bArm2HorzStn5Unhook_25 AT %MX21320.25 : BOOL;
	bArm2HorzStn5Unhook_26 AT %MX21320.26 : BOOL;
	bArm2HorzStn5Unhook_27 AT %MX21320.27 : BOOL;
	bArm2HorzStn5Unhook_28 AT %MX21320.28 : BOOL;
	bArm2HorzStn5Unhook_29 AT %MX21320.29 : BOOL;
	bArm2HorzStn5Unhook_30 AT %MX21320.30 : BOOL;
	bArm2HorzStn5Unhook_31 AT %MX21320.31 : BOOL;

	bArm2HorzStn6Unhook_00 AT %MX21324.0 : BOOL;
	bArm2HorzStn6Unhook_01 AT %MX21324.1 : BOOL;
	bArm2HorzStn6Unhook_02 AT %MX21324.2 : BOOL;
	bArm2HorzStn6Unhook_03 AT %MX21324.3 : BOOL;
	bArm2HorzStn6Unhook_04 AT %MX21324.4 : BOOL;
	bArm2HorzStn6Unhook_05 AT %MX21324.5 : BOOL;
	bArm2HorzStn6Unhook_06 AT %MX21324.6 : BOOL;
	bArm2HorzStn6Unhook_07 AT %MX21324.7 : BOOL;
	bArm2HorzStn6Unhook_08 AT %MX21324.8 : BOOL;
	bArm2HorzStn6Unhook_09 AT %MX21324.9 : BOOL;
	bArm2HorzStn6Unhook_10 AT %MX21324.10 : BOOL;
	bArm2HorzStn6Unhook_11 AT %MX21324.11 : BOOL;
	bArm2HorzStn6Unhook_12 AT %MX21324.12 : BOOL;
	bArm2HorzStn6Unhook_13 AT %MX21324.13 : BOOL;
	bArm2HorzStn6Unhook_14 AT %MX21324.14 : BOOL;
	bArm2HorzStn6Unhook_15 AT %MX21324.15 : BOOL;
	bArm2HorzStn6Unhook_16 AT %MX21324.16 : BOOL;
	bArm2HorzStn6Unhook_17 AT %MX21324.17 : BOOL;
	bArm2HorzStn6Unhook_18 AT %MX21324.18 : BOOL;
	bArm2HorzStn6Unhook_19 AT %MX21324.19 : BOOL;
	bArm2HorzStn6Unhook_20 AT %MX21324.20 : BOOL;
	bArm2HorzStn6Unhook_21 AT %MX21324.21 : BOOL;
	bArm2HorzStn6Unhook_22 AT %MX21324.22 : BOOL;
	bArm2HorzStn6Unhook_23 AT %MX21324.23 : BOOL;
	bArm2HorzStn6Unhook_24 AT %MX21324.24 : BOOL;
	bArm2HorzStn6Unhook_25 AT %MX21324.25 : BOOL;
	bArm2HorzStn6Unhook_26 AT %MX21324.26 : BOOL;
	bArm2HorzStn6Unhook_27 AT %MX21324.27 : BOOL;
	bArm2HorzStn6Unhook_28 AT %MX21324.28 : BOOL;
	bArm2HorzStn6Unhook_29 AT %MX21324.29 : BOOL;
	bArm2HorzStn6Unhook_30 AT %MX21324.30 : BOOL;
	bArm2HorzStn6Unhook_31 AT %MX21324.31 : BOOL;

	bArm2HorzStn7Unhook_00 AT %MX21328.0 : BOOL;
	bArm2HorzStn7Unhook_01 AT %MX21328.1 : BOOL;
	bArm2HorzStn7Unhook_02 AT %MX21328.2 : BOOL;
	bArm2HorzStn7Unhook_03 AT %MX21328.3 : BOOL;
	bArm2HorzStn7Unhook_04 AT %MX21328.4 : BOOL;
	bArm2HorzStn7Unhook_05 AT %MX21328.5 : BOOL;
	bArm2HorzStn7Unhook_06 AT %MX21328.6 : BOOL;
	bArm2HorzStn7Unhook_07 AT %MX21328.7 : BOOL;
	bArm2HorzStn7Unhook_08 AT %MX21328.8 : BOOL;
	bArm2HorzStn7Unhook_09 AT %MX21328.9 : BOOL;
	bArm2HorzStn7Unhook_10 AT %MX21328.10 : BOOL;
	bArm2HorzStn7Unhook_11 AT %MX21328.11 : BOOL;
	bArm2HorzStn7Unhook_12 AT %MX21328.12 : BOOL;
	bArm2HorzStn7Unhook_13 AT %MX21328.13 : BOOL;
	bArm2HorzStn7Unhook_14 AT %MX21328.14 : BOOL;
	bArm2HorzStn7Unhook_15 AT %MX21328.15 : BOOL;
	bArm2HorzStn7Unhook_16 AT %MX21328.16 : BOOL;
	bArm2HorzStn7Unhook_17 AT %MX21328.17 : BOOL;
	bArm2HorzStn7Unhook_18 AT %MX21328.18 : BOOL;
	bArm2HorzStn7Unhook_19 AT %MX21328.19 : BOOL;
	bArm2HorzStn7Unhook_20 AT %MX21328.20 : BOOL;
	bArm2HorzStn7Unhook_21 AT %MX21328.21 : BOOL;
	bArm2HorzStn7Unhook_22 AT %MX21328.22 : BOOL;
	bArm2HorzStn7Unhook_23 AT %MX21328.23 : BOOL;
	bArm2HorzStn7Unhook_24 AT %MX21328.24 : BOOL;
	bArm2HorzStn7Unhook_25 AT %MX21328.25 : BOOL;
	bArm2HorzStn7Unhook_26 AT %MX21328.26 : BOOL;
	bArm2HorzStn7Unhook_27 AT %MX21328.27 : BOOL;
	bArm2HorzStn7Unhook_28 AT %MX21328.28 : BOOL;
	bArm2HorzStn7Unhook_29 AT %MX21328.29 : BOOL;
	bArm2HorzStn7Unhook_30 AT %MX21328.30 : BOOL;
	bArm2HorzStn7Unhook_31 AT %MX21328.31 : BOOL;

	bArm2HorzStn8Unhook_00 AT %MX21332.0 : BOOL;
	bArm2HorzStn8Unhook_01 AT %MX21332.1 : BOOL;
	bArm2HorzStn8Unhook_02 AT %MX21332.2 : BOOL;
	bArm2HorzStn8Unhook_03 AT %MX21332.3 : BOOL;
	bArm2HorzStn8Unhook_04 AT %MX21332.4 : BOOL;
	bArm2HorzStn8Unhook_05 AT %MX21332.5 : BOOL;
	bArm2HorzStn8Unhook_06 AT %MX21332.6 : BOOL;
	bArm2HorzStn8Unhook_07 AT %MX21332.7 : BOOL;
	bArm2HorzStn8Unhook_08 AT %MX21332.8 : BOOL;
	bArm2HorzStn8Unhook_09 AT %MX21332.9 : BOOL;
	bArm2HorzStn8Unhook_10 AT %MX21332.10 : BOOL;
	bArm2HorzStn8Unhook_11 AT %MX21332.11 : BOOL;
	bArm2HorzStn8Unhook_12 AT %MX21332.12 : BOOL;
	bArm2HorzStn8Unhook_13 AT %MX21332.13 : BOOL;
	bArm2HorzStn8Unhook_14 AT %MX21332.14 : BOOL;
	bArm2HorzStn8Unhook_15 AT %MX21332.15 : BOOL;
	bArm2HorzStn8Unhook_16 AT %MX21332.16 : BOOL;
	bArm2HorzStn8Unhook_17 AT %MX21332.17 : BOOL;
	bArm2HorzStn8Unhook_18 AT %MX21332.18 : BOOL;
	bArm2HorzStn8Unhook_19 AT %MX21332.19 : BOOL;
	bArm2HorzStn8Unhook_20 AT %MX21332.20 : BOOL;
	bArm2HorzStn8Unhook_21 AT %MX21332.21 : BOOL;
	bArm2HorzStn8Unhook_22 AT %MX21332.22 : BOOL;
	bArm2HorzStn8Unhook_23 AT %MX21332.23 : BOOL;
	bArm2HorzStn8Unhook_24 AT %MX21332.24 : BOOL;
	bArm2HorzStn8Unhook_25 AT %MX21332.25 : BOOL;
	bArm2HorzStn8Unhook_26 AT %MX21332.26 : BOOL;
	bArm2HorzStn8Unhook_27 AT %MX21332.27 : BOOL;
	bArm2HorzStn8Unhook_28 AT %MX21332.28 : BOOL;
	bArm2HorzStn8Unhook_29 AT %MX21332.29 : BOOL;
	bArm2HorzStn8Unhook_30 AT %MX21332.30 : BOOL;
	bArm2HorzStn8Unhook_31 AT %MX21332.31 : BOOL;

	bArm2HorzStn9Unhook_00 AT %MX21336.0 : BOOL;
	bArm2HorzStn9Unhook_01 AT %MX21336.1 : BOOL;
	bArm2HorzStn9Unhook_02 AT %MX21336.2 : BOOL;
	bArm2HorzStn9Unhook_03 AT %MX21336.3 : BOOL;
	bArm2HorzStn9Unhook_04 AT %MX21336.4 : BOOL;
	bArm2HorzStn9Unhook_05 AT %MX21336.5 : BOOL;
	bArm2HorzStn9Unhook_06 AT %MX21336.6 : BOOL;
	bArm2HorzStn9Unhook_07 AT %MX21336.7 : BOOL;
	bArm2HorzStn9Unhook_08 AT %MX21336.8 : BOOL;
	bArm2HorzStn9Unhook_09 AT %MX21336.9 : BOOL;
	bArm2HorzStn9Unhook_10 AT %MX21336.10 : BOOL;
	bArm2HorzStn9Unhook_11 AT %MX21336.11 : BOOL;
	bArm2HorzStn9Unhook_12 AT %MX21336.12 : BOOL;
	bArm2HorzStn9Unhook_13 AT %MX21336.13 : BOOL;
	bArm2HorzStn9Unhook_14 AT %MX21336.14 : BOOL;
	bArm2HorzStn9Unhook_15 AT %MX21336.15 : BOOL;
	bArm2HorzStn9Unhook_16 AT %MX21336.16 : BOOL;
	bArm2HorzStn9Unhook_17 AT %MX21336.17 : BOOL;
	bArm2HorzStn9Unhook_18 AT %MX21336.18 : BOOL;
	bArm2HorzStn9Unhook_19 AT %MX21336.19 : BOOL;
	bArm2HorzStn9Unhook_20 AT %MX21336.20 : BOOL;
	bArm2HorzStn9Unhook_21 AT %MX21336.21 : BOOL;
	bArm2HorzStn9Unhook_22 AT %MX21336.22 : BOOL;
	bArm2HorzStn9Unhook_23 AT %MX21336.23 : BOOL;
	bArm2HorzStn9Unhook_24 AT %MX21336.24 : BOOL;
	bArm2HorzStn9Unhook_25 AT %MX21336.25 : BOOL;
	bArm2HorzStn9Unhook_26 AT %MX21336.26 : BOOL;
	bArm2HorzStn9Unhook_27 AT %MX21336.27 : BOOL;
	bArm2HorzStn9Unhook_28 AT %MX21336.28 : BOOL;
	bArm2HorzStn9Unhook_29 AT %MX21336.29 : BOOL;
	bArm2HorzStn9Unhook_30 AT %MX21336.30 : BOOL;
	bArm2HorzStn9Unhook_31 AT %MX21336.31 : BOOL;

	bArm2HorzStn10Unhook_00 AT %MX21340.0 : BOOL;
	bArm2HorzStn10Unhook_01 AT %MX21340.1 : BOOL;
	bArm2HorzStn10Unhook_02 AT %MX21340.2 : BOOL;
	bArm2HorzStn10Unhook_03 AT %MX21340.3 : BOOL;
	bArm2HorzStn10Unhook_04 AT %MX21340.4 : BOOL;
	bArm2HorzStn10Unhook_05 AT %MX21340.5 : BOOL;
	bArm2HorzStn10Unhook_06 AT %MX21340.6 : BOOL;
	bArm2HorzStn10Unhook_07 AT %MX21340.7 : BOOL;
	bArm2HorzStn10Unhook_08 AT %MX21340.8 : BOOL;
	bArm2HorzStn10Unhook_09 AT %MX21340.9 : BOOL;
	bArm2HorzStn10Unhook_10 AT %MX21340.10 : BOOL;
	bArm2HorzStn10Unhook_11 AT %MX21340.11 : BOOL;
	bArm2HorzStn10Unhook_12 AT %MX21340.12 : BOOL;
	bArm2HorzStn10Unhook_13 AT %MX21340.13 : BOOL;
	bArm2HorzStn10Unhook_14 AT %MX21340.14 : BOOL;
	bArm2HorzStn10Unhook_15 AT %MX21340.15 : BOOL;
	bArm2HorzStn10Unhook_16 AT %MX21340.16 : BOOL;
	bArm2HorzStn10Unhook_17 AT %MX21340.17 : BOOL;
	bArm2HorzStn10Unhook_18 AT %MX21340.18 : BOOL;
	bArm2HorzStn10Unhook_19 AT %MX21340.19 : BOOL;
	bArm2HorzStn10Unhook_20 AT %MX21340.20 : BOOL;
	bArm2HorzStn10Unhook_21 AT %MX21340.21 : BOOL;
	bArm2HorzStn10Unhook_22 AT %MX21340.22 : BOOL;
	bArm2HorzStn10Unhook_23 AT %MX21340.23 : BOOL;
	bArm2HorzStn10Unhook_24 AT %MX21340.24 : BOOL;
	bArm2HorzStn10Unhook_25 AT %MX21340.25 : BOOL;
	bArm2HorzStn10Unhook_26 AT %MX21340.26 : BOOL;
	bArm2HorzStn10Unhook_27 AT %MX21340.27 : BOOL;
	bArm2HorzStn10Unhook_28 AT %MX21340.28 : BOOL;
	bArm2HorzStn10Unhook_29 AT %MX21340.29 : BOOL;
	bArm2HorzStn10Unhook_30 AT %MX21340.30 : BOOL;
	bArm2HorzStn10Unhook_31 AT %MX21340.31 : BOOL;

	bArm2HorzStn11Unhook_00 AT %MX21344.0 : BOOL;
	bArm2HorzStn11Unhook_01 AT %MX21344.1 : BOOL;
	bArm2HorzStn11Unhook_02 AT %MX21344.2 : BOOL;
	bArm2HorzStn11Unhook_03 AT %MX21344.3 : BOOL;
	bArm2HorzStn11Unhook_04 AT %MX21344.4 : BOOL;
	bArm2HorzStn11Unhook_05 AT %MX21344.5 : BOOL;
	bArm2HorzStn11Unhook_06 AT %MX21344.6 : BOOL;
	bArm2HorzStn11Unhook_07 AT %MX21344.7 : BOOL;
	bArm2HorzStn11Unhook_08 AT %MX21344.8 : BOOL;
	bArm2HorzStn11Unhook_09 AT %MX21344.9 : BOOL;
	bArm2HorzStn11Unhook_10 AT %MX21344.10 : BOOL;
	bArm2HorzStn11Unhook_11 AT %MX21344.11 : BOOL;
	bArm2HorzStn11Unhook_12 AT %MX21344.12 : BOOL;
	bArm2HorzStn11Unhook_13 AT %MX21344.13 : BOOL;
	bArm2HorzStn11Unhook_14 AT %MX21344.14 : BOOL;
	bArm2HorzStn11Unhook_15 AT %MX21344.15 : BOOL;
	bArm2HorzStn11Unhook_16 AT %MX21344.16 : BOOL;
	bArm2HorzStn11Unhook_17 AT %MX21344.17 : BOOL;
	bArm2HorzStn11Unhook_18 AT %MX21344.18 : BOOL;
	bArm2HorzStn11Unhook_19 AT %MX21344.19 : BOOL;
	bArm2HorzStn11Unhook_20 AT %MX21344.20 : BOOL;
	bArm2HorzStn11Unhook_21 AT %MX21344.21 : BOOL;
	bArm2HorzStn11Unhook_22 AT %MX21344.22 : BOOL;
	bArm2HorzStn11Unhook_23 AT %MX21344.23 : BOOL;
	bArm2HorzStn11Unhook_24 AT %MX21344.24 : BOOL;
	bArm2HorzStn11Unhook_25 AT %MX21344.25 : BOOL;
	bArm2HorzStn11Unhook_26 AT %MX21344.26 : BOOL;
	bArm2HorzStn11Unhook_27 AT %MX21344.27 : BOOL;
	bArm2HorzStn11Unhook_28 AT %MX21344.28 : BOOL;
	bArm2HorzStn11Unhook_29 AT %MX21344.29 : BOOL;
	bArm2HorzStn11Unhook_30 AT %MX21344.30 : BOOL;
	bArm2HorzStn11Unhook_31 AT %MX21344.31 : BOOL;

	bArm2HorzStn12Unhook_00 AT %MX21348.0 : BOOL;
	bArm2HorzStn12Unhook_01 AT %MX21348.1 : BOOL;
	bArm2HorzStn12Unhook_02 AT %MX21348.2 : BOOL;
	bArm2HorzStn12Unhook_03 AT %MX21348.3 : BOOL;
	bArm2HorzStn12Unhook_04 AT %MX21348.4 : BOOL;
	bArm2HorzStn12Unhook_05 AT %MX21348.5 : BOOL;
	bArm2HorzStn12Unhook_06 AT %MX21348.6 : BOOL;
	bArm2HorzStn12Unhook_07 AT %MX21348.7 : BOOL;
	bArm2HorzStn12Unhook_08 AT %MX21348.8 : BOOL;
	bArm2HorzStn12Unhook_09 AT %MX21348.9 : BOOL;
	bArm2HorzStn12Unhook_10 AT %MX21348.10 : BOOL;
	bArm2HorzStn12Unhook_11 AT %MX21348.11 : BOOL;
	bArm2HorzStn12Unhook_12 AT %MX21348.12 : BOOL;
	bArm2HorzStn12Unhook_13 AT %MX21348.13 : BOOL;
	bArm2HorzStn12Unhook_14 AT %MX21348.14 : BOOL;
	bArm2HorzStn12Unhook_15 AT %MX21348.15 : BOOL;
	bArm2HorzStn12Unhook_16 AT %MX21348.16 : BOOL;
	bArm2HorzStn12Unhook_17 AT %MX21348.17 : BOOL;
	bArm2HorzStn12Unhook_18 AT %MX21348.18 : BOOL;
	bArm2HorzStn12Unhook_19 AT %MX21348.19 : BOOL;
	bArm2HorzStn12Unhook_20 AT %MX21348.20 : BOOL;
	bArm2HorzStn12Unhook_21 AT %MX21348.21 : BOOL;
	bArm2HorzStn12Unhook_22 AT %MX21348.22 : BOOL;
	bArm2HorzStn12Unhook_23 AT %MX21348.23 : BOOL;
	bArm2HorzStn12Unhook_24 AT %MX21348.24 : BOOL;
	bArm2HorzStn12Unhook_25 AT %MX21348.25 : BOOL;
	bArm2HorzStn12Unhook_26 AT %MX21348.26 : BOOL;
	bArm2HorzStn12Unhook_27 AT %MX21348.27 : BOOL;
	bArm2HorzStn12Unhook_28 AT %MX21348.28 : BOOL;
	bArm2HorzStn12Unhook_29 AT %MX21348.29 : BOOL;
	bArm2HorzStn12Unhook_30 AT %MX21348.30 : BOOL;
	bArm2HorzStn12Unhook_31 AT %MX21348.31 : BOOL;


(* xxxxxxxxxxxxxxxxxxxxxxxxxxxxxxxxxxxxxxx Vert xxxxxxxxxxxxxxxxxxxxxxxxxxxxxxxxxxxxxxx*)
(*========= Up BOOL LINK with %MX26000-MX26099 =========*)

	bArm2VertLD1Up_00 AT %MX26052.0 : BOOL;
	bArm2VertLD1Up_01 AT %MX26052.1 : BOOL;
	bArm2VertLD1Up_02 AT %MX26052.2 : BOOL;
	bArm2VertLD1Up_03 AT %MX26052.3 : BOOL;
	bArm2VertLD1Up_04 AT %MX26052.4 : BOOL;
	bArm2VertLD1Up_05 AT %MX26052.5 : BOOL;
	bArm2VertLD1Up_06 AT %MX26052.6 : BOOL;
	bArm2VertLD1Up_07 AT %MX26052.7 : BOOL;
	bArm2VertLD1Up_08 AT %MX26052.8 : BOOL;
	bArm2VertLD1Up_09 AT %MX26052.9 : BOOL;
	bArm2VertLD1Up_10 AT %MX26052.10 : BOOL;
	bArm2VertLD1Up_11 AT %MX26052.11 : BOOL;
	bArm2VertLD1Up_12 AT %MX26052.12 : BOOL;
	bArm2VertLD1Up_13 AT %MX26052.13 : BOOL;
	bArm2VertLD1Up_14 AT %MX26052.14 : BOOL;
	bArm2VertLD1Up_15 AT %MX26052.15 : BOOL;
	bArm2VertLD1Up_16 AT %MX26052.16 : BOOL;
	bArm2VertLD1Up_17 AT %MX26052.17 : BOOL;
	bArm2VertLD1Up_18 AT %MX26052.18 : BOOL;
	bArm2VertLD1Up_19 AT %MX26052.19 : BOOL;
	bArm2VertLD1Up_20 AT %MX26052.20 : BOOL;
	bArm2VertLD1Up_21 AT %MX26052.21 : BOOL;
	bArm2VertLD1Up_22 AT %MX26052.22 : BOOL;
	bArm2VertLD1Up_23 AT %MX26052.23 : BOOL;
	bArm2VertLD1Up_24 AT %MX26052.24 : BOOL;
	bArm2VertLD1Up_25 AT %MX26052.25 : BOOL;
	bArm2VertLD1Up_26 AT %MX26052.26 : BOOL;
	bArm2VertLD1Up_27 AT %MX26052.27 : BOOL;
	bArm2VertLD1Up_28 AT %MX26052.28 : BOOL;
	bArm2VertLD1Up_29 AT %MX26052.29 : BOOL;
	bArm2VertLD1Up_30 AT %MX26052.30 : BOOL;
	bArm2VertLD1Up_31 AT %MX26052.31 : BOOL;

